(* Logix 5000 project; controller RN21_Architecture 1769-L16ER-BB1B rev 35.11; software revision 35.00; part 3 of 9 *)

ADD_ON_INSTRUCTION AOI_TBC   (* revision 1.0 *)
VAR_INPUT
   FBI_AuditPLC_UID : DINT; {access None, required}
END_VAR
VAR_OUTPUT
   FBO_TBCAuditPLC_UID : DINT; {required}
END_VAR
VAR_INPUT
   FBI_AlarmPLC_UID : DINT; {required}
END_VAR
VAR_OUTPUT
   FBO_TBCAlarmPLC_UID : DINT; {required}
END_VAR
VAR_INPUT
   FBI_RecipePLC_UID : DINT; {required}
END_VAR
VAR_OUTPUT
   FBO_TBCRecipePLC_UID : DINT; {required}
END_VAR
VAR_INPUT
   FBI_UMPLC_UID : DINT; {required}
END_VAR
VAR_OUTPUT
   FBO_TBCUMPLC_UID : DINT; {required}
END_VAR
VAR_INPUT
   FBI_BatchPLC_UID : DINT; {required}
END_VAR
VAR_OUTPUT
   FBO_TBCBatchPLC_UID : DINT; {required}
END_VAR
VAR_INPUT
   FBI_AuditServer_UID : DINT; {required}
END_VAR
VAR_OUTPUT
   FBO_TBCAuditServer_UID : DINT; {required}
END_VAR
VAR_INPUT
   FBI_AlarmServer_UID : DINT; {required}
END_VAR
VAR_OUTPUT
   FBO_TBCAlarmServer_UID : DINT; {required}
END_VAR
VAR_INPUT
   FBI_RecipeServer_UID : DINT; {required}
END_VAR
VAR_OUTPUT
   FBO_TBCRecipeServer_UID : DINT; {required}
END_VAR
VAR_INPUT
   FBI_UMServer_UID : DINT; {required}
END_VAR
VAR_OUTPUT
   FBO_TBCUMServer_UID : DINT; {required}
END_VAR
VAR_INPUT
   FBI_BatchServer_UID : DINT; {required}
END_VAR
VAR_OUTPUT
   FBO_TBCBatchServer_UID : DINT; {required}
   FBO_TBCProcessServer_UID : DINT; {required}
END_VAR
VAR_INPUT
   FBI_ProcessServer_UID : DINT; {required}
   FBI_ProcessPLC_UID : DINT; {required}
END_VAR
VAR_OUTPUT
   FBO_TBCProcessPLC_UID : DINT; {required}
END_VAR
VAR_IN_OUT
   FBIO_Batch_Trigger : BOOL; {required}
   FBIO_UM_Trigger : BOOL; {required}
   FBIO_Process_Trigger : BOOL; {required}
   FBIO_Recipe_Trigger : BOOL; {required}
   FBIO_Audit_Trigger : BOOL; {required}
   FBIO_Alarm_Trigger : BOOL; {required}
END_VAR
VAR_OUTPUT
   FBO_TBCPosition : DINT; {required}
   TBCUID : DINT; {required}
END_VAR
VAR_IN_OUT
   FBI_TBCServerAlarm_Trig : BOOL; {required}
   FBI_TBCServerProces_Trig : BOOL; {required}
   FBI_TBCServerAudit_Trig : BOOL; {required}
   FBI_TBCServerBatch_Trig : BOOL; {required}
   FBI_TBCServerRecipe_Trig : BOOL; {required}
   FBI_TBCServerUM_Trig : BOOL; {required}
END_VAR
VAR
   TMR_TBCTrigger : TIMER := (PRE := 60000); {access None}
   CTU_TBCUID : COUNTER := (PRE := 32767); {access None}
   FBL_TBCPosition : DINT; {access None}
   TMRTBC_AlmTrigRst : TIMER := (PRE := 10000); {access None}
   TMRTBC_UMTrigRst : TIMER := (PRE := 10000); {access None}
   TMRTBC_ProcessTrigRst : TIMER := (PRE := 10000); {access None}
   TMRTBC_AuditTrigRst : TIMER := (PRE := 10000); {access None}
   TMRTBC_BatchTrigRst : TIMER := (PRE := 10000); {access None}
   TMRTBC_RecipeTrigRst : TIMER := (PRE := 10000); {access None}
END_VAR

ROUTINE Logic   (* ladder *)
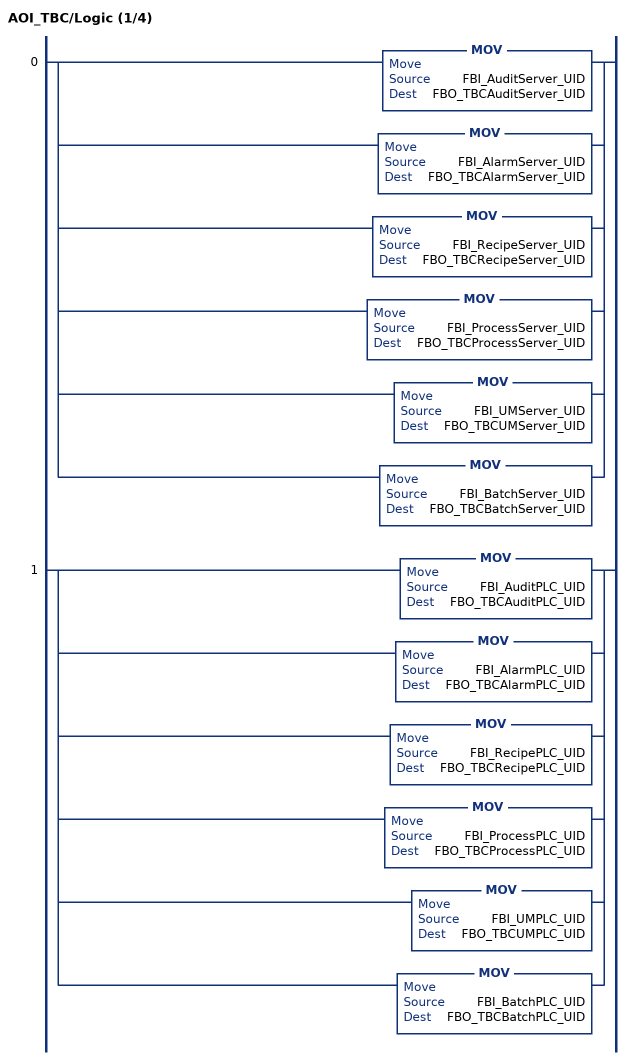
   0: [MOV(FBI_AuditServer_UID,FBO_TBCAuditServer_UID) ,MOV(FBI_AlarmServer_UID,FBO_TBCAlarmServer_UID) ,MOV(FBI_RecipeServer_UID,FBO_TBCRecipeServer_UID) ,MOV(FBI_ProcessServer_UID,FBO_TBCProcessServer_UID) ,MOV(FBI_UMServer_UID,FBO_TBCUMServer_UID) ,MOV(FBI_BatchServer_UID,FBO_TBCBatchServer_UID) ];
   1: [MOV(FBI_AuditPLC_UID,FBO_TBCAuditPLC_UID) ,MOV(FBI_AlarmPLC_UID,FBO_TBCAlarmPLC_UID) ,MOV(FBI_RecipePLC_UID,FBO_TBCRecipePLC_UID) ,MOV(FBI_ProcessPLC_UID,FBO_TBCProcessPLC_UID) ,MOV(FBI_UMPLC_UID,FBO_TBCUMPLC_UID) ,MOV(FBI_BatchPLC_UID,FBO_TBCBatchPLC_UID) ];
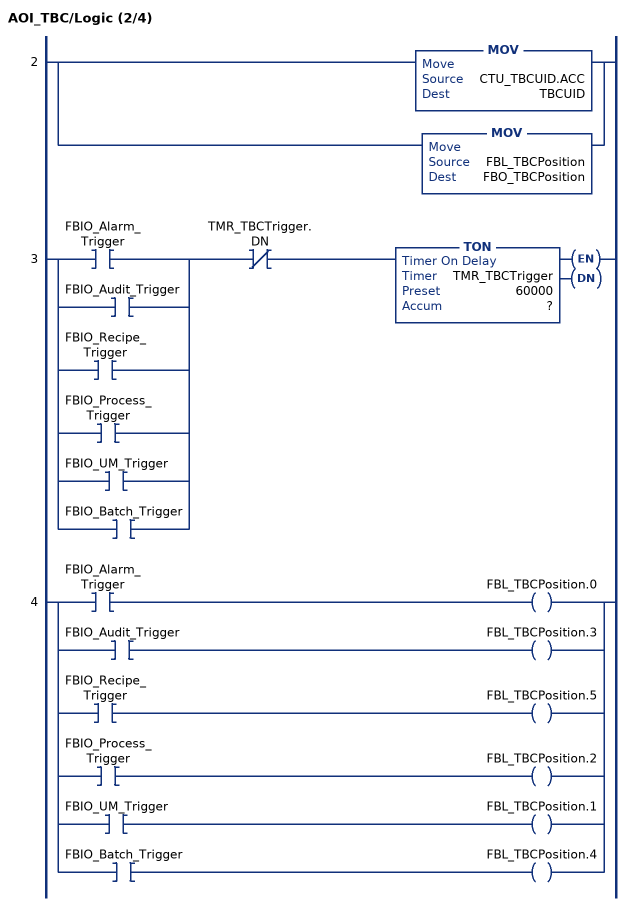
   2: [MOV(CTU_TBCUID.ACC,TBCUID) ,MOV(FBL_TBCPosition,FBO_TBCPosition) ];
   3: [XIC(FBIO_Alarm_Trigger) ,XIC(FBIO_Audit_Trigger) ,XIC(FBIO_Recipe_Trigger) ,XIC(FBIO_Process_Trigger) ,XIC(FBIO_UM_Trigger) ,XIC(FBIO_Batch_Trigger) ]XIO(TMR_TBCTrigger.DN)TON(TMR_TBCTrigger,?,?);
   4: [XIC(FBIO_Alarm_Trigger) OTE(FBL_TBCPosition.0) ,XIC(FBIO_Audit_Trigger) OTE(FBL_TBCPosition.3) ,XIC(FBIO_Recipe_Trigger) OTE(FBL_TBCPosition.5) ,XIC(FBIO_Process_Trigger) OTE(FBL_TBCPosition.2) ,XIC(FBIO_UM_Trigger) OTE(FBL_TBCPosition.1) ,XIC(FBIO_Batch_Trigger) OTE(FBL_TBCPosition.4) ];
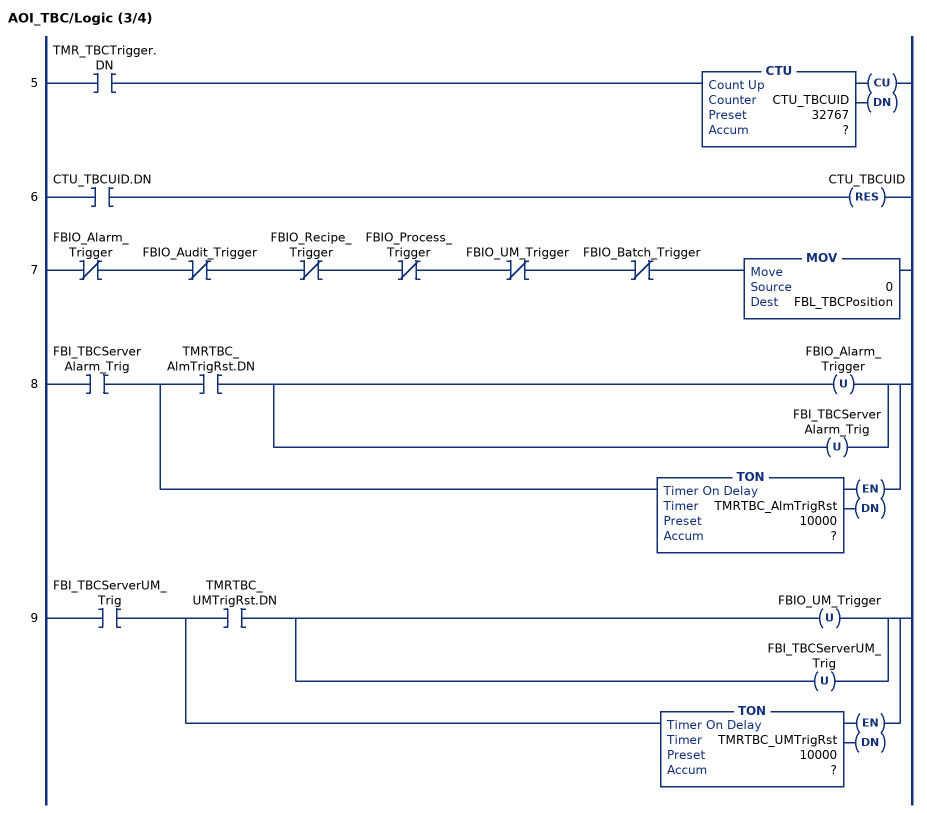
   5: XIC(TMR_TBCTrigger.DN)CTU(CTU_TBCUID,?,?);
   6: XIC(CTU_TBCUID.DN)RES(CTU_TBCUID);
   7: XIO(FBIO_Alarm_Trigger)XIO(FBIO_Audit_Trigger)XIO(FBIO_Recipe_Trigger)XIO(FBIO_Process_Trigger)XIO(FBIO_UM_Trigger)XIO(FBIO_Batch_Trigger)MOV(0,FBL_TBCPosition);
   8: XIC(FBI_TBCServerAlarm_Trig)[XIC(TMRTBC_AlmTrigRst.DN) [OTU(FBIO_Alarm_Trigger) ,OTU(FBI_TBCServerAlarm_Trig) ] ,TON(TMRTBC_AlmTrigRst,?,?) ];
   9: XIC(FBI_TBCServerUM_Trig)[XIC(TMRTBC_UMTrigRst.DN) [OTU(FBIO_UM_Trigger) ,OTU(FBI_TBCServerUM_Trig) ] ,TON(TMRTBC_UMTrigRst,?,?) ];
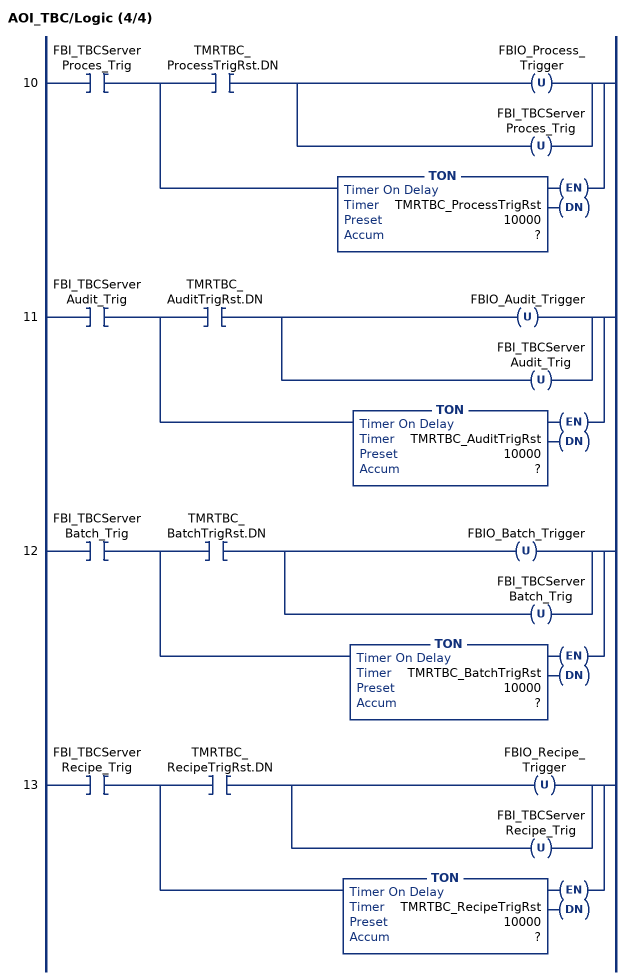
   10: XIC(FBI_TBCServerProces_Trig)[XIC(TMRTBC_ProcessTrigRst.DN) [OTU(FBIO_Process_Trigger) ,OTU(FBI_TBCServerProces_Trig) ] ,TON(TMRTBC_ProcessTrigRst,?,?) ];
   11: XIC(FBI_TBCServerAudit_Trig)[XIC(TMRTBC_AuditTrigRst.DN) [OTU(FBIO_Audit_Trigger) ,OTU(FBI_TBCServerAudit_Trig) ] ,TON(TMRTBC_AuditTrigRst,?,?) ];
   12: XIC(FBI_TBCServerBatch_Trig)[XIC(TMRTBC_BatchTrigRst.DN) [OTU(FBIO_Batch_Trigger) ,OTU(FBI_TBCServerBatch_Trig) ] ,TON(TMRTBC_BatchTrigRst,?,?) ];
   13: XIC(FBI_TBCServerRecipe_Trig)[XIC(TMRTBC_RecipeTrigRst.DN) [OTU(FBIO_Recipe_Trigger) ,OTU(FBI_TBCServerRecipe_Trig) ] ,TON(TMRTBC_RecipeTrigRst,?,?) ];
END_ROUTINE
END_ADD_ON_INSTRUCTION

VAR_GLOBAL   (* controller tags *)
   ALM_TriggerId : BOOL := 1;
   ALM_UniqueNum : DINT := 300;
   ALMSer : UDT_Alarm := (ALM_YearValue := 2026, ALM_MonthValue := 3, ALM_DayValue := 3, ALM_HourValue := 18, ALM_MinuteValue := 48, ALM_SecondValue := 11, ALM_AlarmId1 := 3);
   AUD_TriggerId : BOOL;
   AUD_UniqueNum : DINT := 911;
   AUDSer : UDT_Audit := (AUD_YearValue := 2026, AUD_MonthValue := 3, AUD_DayValue := 3, AUD_HourValue := 12, AUD_SecondValue := 30, AUD_ActionId := 6009, AUD_NewValue := 389.0, AUD_AppUserId := 'EMGUSER');
   BACK_BATCH_NO : STRING := 'ee3';
   BACK_BatchStartACK : DINT;
   BACK_LOT_NO : STRING := 'uuuu';
   BMAN_BatchUniqueId : DINT := 63;
   BMAN_TriggerBit : BOOL;
   BMANSer : UDT_Batch := (BMAN_YearValue := 2026, BMAN_MonthValue := 3, BMAN_DayValue := 2, BMAN_HourValue := 17, BMAN_MinuteValue := 33, BMAN_SecondValue := 37, BMAN_BatchStatus := 2, BMAN_BATCH_RECIPENAME := 'CLST5000', BMAN_LOT_NO := 'lot1', BMAN_PRODUCT_CODE := 'Compa', BMAN_PRODUCT_NAME := 'Compa', BMAN_BATCH_NO := 'Tes');
   Controller_FirstScan : BOOL;
   DummyBit : BOOL;
   EmergencyLoginActivated_Bit : BOOL := 1;
   EmergencyUserIDEqual : BOOL;
   EmergencyUserPaswdEqual : BOOL;
   FCI_C1PAUSE_RELEASE : BOOL;
   FCI_C1START : BOOL;
   FCI_C1STOP : BOOL;
   FCO_C1STARTED : BOOL;
   HB_HEART_BEAT : BOOL := 1;
   LBSer : UDT_Login := (LOGIN_YearValue := 2026, LOGIN_MonthValue := 3, LOGIN_DayValue := 4, LOGIN_HourValue := 10, LOGIN_MinuteValue := 9, LOGIN_SecondValue := 53, LOGIN_Reason := 28, LOGIN_LoginReason := -1, LOGIN_AppUserId := 'Navin$00$00');
   LOGIN_TriggerId : BOOL := 1;
   LOGIN_UniqueNum : DINT := 570;
   PDL_Trigger : BOOL;
   PDL_UID : DINT := 701;
   PDLSer : UDT_Process := (PDL_Year := 2026, PDL_Month := 1, PDL_Date := 13, PDL_Hour := 17, PDL_Minute := 22, PDL_Second := 27, PDL_CYCLEID := 2, PDL_ProcessData[0] := 3.0, PDL_ProcessData[1] := 5.0, PDL_ProcessData[2] := 5.0, PDL_ProcessData[3] := 6.0, PDL_ProcessData[4] := 2.2, PDL_ProcessData[5] := 11.2, PDL_ProcessData[6] := 11.9, PDL_ProcessData[7] := 41.5);
   RM_RecipeAck : DINT := 2;
   RM_RecipeCode : STRING := 'CLST5000';
   RN21_BACK_BatchSize : REAL := 51.02;
   RN21_BACK_ProductCode : STRING := 'AKHBJ';
   RN21_BACK_ProductName : STRING := 'AEBJH';
   RN21_EmgUserID : STRING := 'EMGUSER';
   RN21_FirstScan : BOOL;
   RN21_HMIScrennControl : DINT;
   RN21_PDLMainONS : BOOL;
   RN21_UM_EmgPSWD : STRING := 'EMG1234';
   RP_Trigger : BOOL;
   RP_UID : DINT := 31;
   RPSer : UDT_Recipe := (RP_Year := 2026, RP_Month := 1, RP_Date := 12, RP_Hour := 10, RP_Minute := 57, RP_Second := 54, RP_RecipeData1[0] := 10.0, RP_RecipeData1[1] := 11.1, RP_RecipeData1[2] := 22.2, RP_RecipeData1[3] := 33.3, RP_RecipeData1[4] := 44.4, RP_RecipeData1[5] := 55.5, RP_RecipeData1[6] := 66.6, RP_RecipeData1[7] := 77.7, RP_RecipeData1[8] := 88.8, RP_RecipeData1[9] := 99.9, RP_RecipeData2[0] := 10, RP_RecipeData2[1] := 20, RP_RecipeData2[2] := 30, RP_RecipeData2[3] := 40, RP_RecipeData2[4] := 50, RP_RecipeData2[5] := 60, RP_RecipeData2[6] := 70, RP_RecipeData2[7] := 80, RP_RecipeData2[8] := 90, RP_RecipeData2[9] := 100);
   RTC_DATE_AND_TIME_UNLATCH_DELAY : COUNTER := (PRE := 2);
   RTC_DAY : DINT := 3;
   RTC_HOUR : DINT := 12;
   RTC_MINUTE : DINT := 23;
   RTC_MONTH : DINT := 3;
   RTC_SAVE_DATE_AND_TIME : BOOL;
   RTC_SECONDS : DINT := 14;
   RTC_UniqueId : DINT := 97;
   RTC_YEAR : DINT := 2026;
   ServerRTC : DINT[8] := ([0] := 2026, [1] := 3, [2] := 25, [3] := 5, [4] := 43, [5] := 2);
   TBC_ALARMBLOCK_PLCUID : DINT := 304;
   TBC_ALARMBLOCK_SERVERUID : DINT := 300;
   TBC_ALARMBLOCK_TRIGGER : BOOL;
   TBC_AUDITBLOCK_PLCUID : DINT := 911;
   TBC_AUDITBLOCK_SERVERUID : DINT := 911;
   TBC_AUDITBLOCK_TRIGGER : BOOL;
   TBC_BATCHMGMTBLOCK_PLCUID : DINT;
   TBC_BATCHMGMTBLOCK_SERVERUID : DINT := 63;
   TBC_BATCHMGMTBLOCK_TRIGGER : BOOL;
   TBC_POSITION : DINT := 3;
   TBC_PROCESSBLOCK_PLCUID : DINT := 701;
   TBC_PROCESSBLOCK_SERVERUID : DINT := 701;
   TBC_PROCESSBLOCK_TRIGGER : BOOL;
   TBC_RECIPEBLOCK_PLCUID : DINT := 31;
   TBC_RECIPEBLOCK_SERVERUID : DINT := 31;
   TBC_RECIPEBLOCK_TRIGGER : BOOL;
   TBC_UID : DINT;
   TBC_UMBLOCK_PLCUID : DINT := 581;
   TBC_UMBLOCK_SERVERUID : DINT := 570;
   TBC_UMBLOCK_TRIGGER : BOOL;
   UM_ACT : DINT;
   UM_Confirmation_Bit : BOOL;
   UM_EXPIRY : DINT;
   UM_EXPIRY_DAYS : DINT := 78;
   UM_lockoutDurationLeft : DINT;
   UM_LVL : DINT;
   UM_NoOfAttempts : DINT := 5;
   UM_PWD : STRING := '0';
   UM_Status : DINT;
   UM_UID : STRING := '0';
   UM_UID_OUT : STRING := 'Navin';
   UM_UniqueID : DINT := 520;
END_VAR

PROGRAM MainProgram   (* main routine MainRoutine *)
VAR
   ALMSrc : UDT_Alarm := (ALM_YearValue := 2026, ALM_MonthValue := 3, ALM_DayValue := 4, ALM_HourValue := 14, ALM_MinuteValue := 57, ALM_SecondValue := 10, ALM_AlarmId1 := 1);
   ALMSrc_UniqueNum : DINT := 304;
   ANM_C1Pause_Release : BOOL;
   ANM_C1StartReq : BOOL;
   ANM_C1StopReq_Auto : BOOL;
   ANM_C1StopReq_HMI : BOOL;
   ANM_C2Pause_Release : BOOL;
   ANM_C2StartReq : BOOL;
   ANM_C2StopReq_Auto : BOOL;
   ANM_C2StopReq_HMI : BOOL;
   ANM_C3Pause_Release : BOOL;
   ANM_C3StartReq : BOOL;
   ANM_C3StopReq_Auto : BOOL;
   ANM_C3StopReq_HMI : BOOL;
   ANM_C4Pause_Release : BOOL;
   ANM_C4StartReq : BOOL;
   ANM_C4StopReq_Auto : BOOL;
   ANM_C4StopReq_HMI : BOOL;
   ANM_C5Pause_Release : BOOL;
   ANM_C5StartReq : BOOL;
   ANM_C5StopReq_Auto : BOOL;
   ANM_C5StopReq_HMI : BOOL;
   ANM_CStopReq_Alarm : BOOL;
   ANM_CycleReset : BOOL;
   AUDSrc : UDT_Audit := (AUD_YearValue := 2026, AUD_MonthValue := 3, AUD_DayValue := 4, AUD_HourValue := 14, AUD_MinuteValue := 57, AUD_SecondValue := 10, AUD_ActionId := 6009, AUD_NewValue := 389.0, AUD_AppUserId := 'EMGUSER');
   AUDSrc_UniqueNum : DINT := 911;
   BIT_RESET_TMR : TIMER := (PRE := 5000);
   BMANSrc : UDT_Batch := (BMAN_YearValue := 2026, BMAN_MonthValue := 3, BMAN_DayValue := 4, BMAN_HourValue := 14, BMAN_MinuteValue := 57, BMAN_SecondValue := 10, BMAN_BatchStatus := 2, BMAN_BATCH_RECIPENAME := 'CLS');
   BMANSrc_UniqueNum : DINT := 63;
   Delformovingupdatedtimertonewpswd : TIMER := (PRE := 2000);
   EmgLoginDn : BOOL;
   EnableInactivity : DINT;
   ExpDays_NoofattemptsLeft_visb : BOOL;
   ExpDays_NoofattemptsLeft_visbility : BOOL := 1;
   ExpiryDays_MovFrmSrv : DINT := 78;
   FC_ALM_Arch : AOI_ALM_Arch := (FBI_PLCServerCommFailed := 1);
   FC_ALM_DC : AOI_ALM_DataCapture[160] := ([0].FBI_AlarmTag := 1, [0].FBO_AlarmPosID := 1);
   FC_AUD_Arch : AOI_AUD_Arch := (FBI_PLCServerCommFailed := 1);
   FC_BMAN_Arch : AOI_BMAN_Arch := (FBI_PLCServerCommFailed := 1);
   FC_LB_Arch : AOI_LOGIN_Arch := (FBI_PLCServerCommFailed := 1);
   FC_PDL_Arch : AOI_PDL_Arch := (FBI_PLCServerCommFailed := 1);
   FC_PDL_DC : AOI_PDL_DataCapture[10] := ([0].FBI_IsPrintIntervalReq := 1, [0].FBI_PrintInterval := 60, [0].FBI_OneSecTrig := 1, [0].FBI_Enable := 1, [0].FBO_Active := 1, [1].FBI_IsPrintIntervalReq := 1, [1].FBI_PrintInterval := 60, [1].FBI_OneSecTrig := 1, [1].FBI_Enable := 1, [1].FBO_Active := 1, [2].FBI_IsPrintIntervalReq := 1, [2].FBI_PrintInterval := 60, [2].FBI_OneSecTrig := 1, [2].FBI_Enable := 1, [2].FBO_Active := 1, [3].FBI_IsPrintIntervalReq := 1, [3].FBI_PrintInterval := 60, [3].FBI_OneSecTrig := 1, [3].FBI_Enable := 1, [3].FBO_Active := 1, [4].FBI_IsPrintIntervalReq := 1, [4].FBI_PrintInterval := 60, [4].FBI_OneSecTrig := 1, [4].FBI_Enable := 1, [4].FBO_Active := 1);
   FC_RP_Arch : AOI_RP_Arch := (FBI_PLCServerCommFailed := 1);
   FC_TBC : AOI_TBC := (FBI_AuditPLC_UID := 911, FBO_TBCAuditPLC_UID := 911, FBI_AlarmPLC_UID := 304, FBO_TBCAlarmPLC_UID := 304, FBI_RecipePLC_UID := 31, FBO_TBCRecipePLC_UID := 31, FBI_UMPLC_UID := 581, FBO_TBCUMPLC_UID := 581, FBI_BatchPLC_UID := 63, FBO_TBCBatchPLC_UID := 63, FBI_AuditServer_UID := 911, FBO_TBCAuditServer_UID := 911, FBI_AlarmServer_UID := 300, FBO_TBCAlarmServer_UID := 300, FBI_RecipeServer_UID := 31, FBO_TBCRecipeServer_UID := 31, FBI_UMServer_UID := 570, FBO_TBCUMServer_UID := 570, FBI_BatchServer_UID := 63, FBO_TBCBatchServer_UID := 63, FBO_TBCProcessServer_UID := 701, FBI_ProcessServer_UID := 701, FBI_ProcessPLC_UID := 701, FBO_TBCProcessPLC_UID := 701, FBO_TBCPosition := 3, TBCUID := 2932);
   FCI_ALARM : BOOL;
   FCI_AlarmReset : BOOL;
   FCI_ALMDataLogTrig : BOOL;
   FCI_AUDDataLogTrig : BOOL;
   FCI_BMANDataLogTrig : BOOL;
   FCI_C1COMPLETED : BOOL;
   FCI_C2COMPLETED : BOOL;
   FCI_C2PAUSE_RELEASE : BOOL;
   FCI_C2START : BOOL;
   FCI_C2STOP : BOOL;
   FCI_C3COMPLETED : BOOL;
   FCI_C3PAUSE_RELEASE : BOOL;
   FCI_C3START : BOOL;
   FCI_C3STOP : BOOL;
   FCI_C4COMPLETED : BOOL;
   FCI_C4PAUSE_RELEASE : BOOL;
   FCI_C4START : BOOL;
   FCI_C4STOP : BOOL;
   FCI_C5COMPLETED : BOOL;
   FCI_C5PAUSE_RELEASE : BOOL;
   FCI_C5STARTED : BOOL;
   FCI_C5STOP : BOOL;
   FCI_LBDataLogTrig : BOOL;
   FCI_PDLDataLogTrig : BOOL;
   FCI_PrintInterval : INT := 60;
   FCI_PROCESSRESET : BOOL;
   FCI_RPDataLogTrig : BOOL;
   FCO_ALMTrig : DINT[5];
   FCO_C1CMPLTSTSMOVTRIG : BOOL;
   FCO_C1PAUSED : BOOL;
   FCO_C1PAUSEDSTSMOVTRIG : BOOL;
   FCO_C1RELEASEDSTSMOVTRIG : BOOL;
   FCO_C1RUNNINGSTSMOVTRIG : BOOL;
   FCO_C1STOPEDALMSTSMOVTRIG : BOOL;
   FCO_C1STOPEDSTSMOVTRIG : BOOL;
   FCO_C2CMPLTSTSMOVTRIG : BOOL;
   FCO_C2PAUSED : BOOL;
   FCO_C2PAUSEDSTSMOVTRIG : BOOL;
   FCO_C2RELEASEDSTSMOVTRIG : BOOL;
   FCO_C2RUNNINGSTSMOVTRIG : BOOL;
   FCO_C2STARTED : BOOL;
   FCO_C2STOPEDALMSTSMOVTRIG : BOOL;
   FCO_C2STOPEDSTSMOVTRIG : BOOL;
   FCO_C3CMPLTSTSMOVTRIG : BOOL;
   FCO_C3PAUSED : BOOL;
   FCO_C3PAUSEDSTSMOVTRIG : BOOL;
   FCO_C3RELEASEDSTSMOVTRIG : BOOL;
   FCO_C3RUNNINGSTSMOVTRIG : BOOL;
   FCO_C3STARTED : BOOL;
   FCO_C3STOPEDALMSTSMOVTRIG : BOOL;
   FCO_C3STOPEDSTSMOVTRIG : BOOL;
   FCO_C4CMPLTSTSMOVTRIG : BOOL;
   FCO_C4PAUSED : BOOL;
   FCO_C4PAUSEDSTSMOVTRIG : BOOL;
   FCO_C4RELEASEDSTSMOVTRIG : BOOL;
   FCO_C4RUNNINGSTSMOVTRIG : BOOL;
   FCO_C4STARTED : BOOL;
   FCO_C4STOPEDALMSTSMOVTRIG : BOOL;
   FCO_C4STOPEDSTSMOVTRIG : BOOL;
   FCO_C5CMPLTSTSMOVTRIG : BOOL;
   FCO_C5PAUSED : BOOL;
   FCO_C5PAUSEDSTSMOVTRIG : BOOL;
   FCO_C5RELEASEDSTSMOVTRIG : BOOL;
   FCO_C5RUNNINGSTSMOVTRIG : BOOL;
   FCO_C5STARTED : BOOL;
   FCO_C5STOPEDALARMSTSMOVTRIG : BOOL;
   FCO_C5STOPEDSTSMOVTRIG : BOOL;
   HMI_ChangePswd : BOOL;
   HMI_CONTROL_SCREEN : DINT;
   HmiCurrentScreen : DINT;
   HMIOLDSCREENVALUE : DINT;
   HMISCREEN : BOOL;
   HMISCREENCHANGED : BOOL;
   inactivity_in_minutes : DINT;
   inactivity_time : DINT := 5;
   INTERNAL_RN21_HB_PLC2ServerCommFailed : BOOL;
   INTERNAL_RN21_PLC2HMICommFailed : BOOL;
   InvalidBit : BOOL;
   LBSrc : UDT_Login := (LOGIN_YearValue := 2026, LOGIN_MonthValue := 3, LOGIN_DayValue := 4, LOGIN_HourValue := 14, LOGIN_MinuteValue := 57, LOGIN_SecondValue := 10, LOGIN_Reason := -1, LOGIN_LoginReason := -32768, LOGIN_AppUserId := 'EMGUSER');
   LBSrc_UniqueNum : DINT := 581;
   Lockout_Visb : BOOL;
   Logged_User : STRING := '0';
   LoginDNDel : TIMER := (PRE := 5000);
   MaskTag : STRING := '************';
   MaskTag1 : STRING := '0';
   New_Pswd : STRING := '0';
   New_Pswd_mask : STRING := '************';
   New_Pswd_mask1 : STRING := '0';
   Password_Change_Yes_Button_In_HMI : BOOL;
   PDLSrc : UDT_Process := (PDL_Year := 2026, PDL_Month := 3, PDL_Date := 4, PDL_Hour := 14, PDL_Minute := 57, PDL_Second := 10, PDL_CYCLEID := 2, PDL_ProcessData[0] := 3.0, PDL_ProcessData[1] := 5.0, PDL_ProcessData[2] := 5.0, PDL_ProcessData[3] := 6.0, PDL_ProcessData[4] := 2.2, PDL_ProcessData[5] := 11.2, PDL_ProcessData[6] := 11.9, PDL_ProcessData[7] := 41.5);
   PDLSrc_PDL_UID : DINT := 701;
   PLC_HMI_CommTag : BOOL;
   PLC_RTC : DINT[7] := ([0] := 2026, [1] := 3, [2] := 4, [3] := 14, [4] := 57, [5] := 10, [6] := 68182);
   PrintIntervalReq : BOOL := 1;
   Pswd_UpadatedSuccessfully : BOOL;
   pwdons : BOOL;
   RecipeEntryFloat : REAL[20] := ([0] := 10.0, [1] := 11.1, [2] := 22.2, [3] := 33.3, [4] := 44.4, [5] := 55.5, [6] := 66.6, [7] := 77.7, [8] := 88.8, [9] := 99.9, [10] := 100.0, [11] := 111.1, [12] := 222.2, [13] := 333.3, [14] := 444.4, [15] := 555.5, [16] := 666.6, [17] := 777.7, [18] := 888.8, [19] := 12.2);
   RecipeEntryInt : INT[11] := ([0] := 10, [1] := 20, [2] := 30, [3] := 40, [4] := 50, [5] := 60, [6] := 70, [7] := 80, [8] := 90, [9] := 100, [10] := 110);
   Remaining_time : DINT;
   remaining_time_compareTag : DINT;
   RN21_AUD_BAMTrig : DINT[5];
   RN21_AUD_BAT_NTrig : DINT[4];
   RN21_AUD_BAT_PTrig : DINT[4];
   RN21_AUD_CompVal : REAL[305] := ([0] := 350.0, [1] := 700.0, [2] := 360.0, [3] := 61.0, [4] := 893.0, [5] := 183.0, [6] := 947.0, [7] := 317.0, [8] := 412.0, [9] := 389.0);
   RN21_AUD_HoldVal : REAL[305] := ([0] := 300.0, [1] := 600.0);
   RN21_AUD_NE_ONS : BOOL[320];
   RN21_AUD_NEG_ONS : BOOL[128];
   RN21_AUD_NETrig : DINT[11];
   RN21_AUD_POS_ONS : BOOL[128];
   RN21_AUDBAM_ONS : BOOL[128];
   RN21_AutoLogedOut : BOOL;
   RN21_BACK_BatchDataStatus : BOOL;   // BATCH START ACKNOWLEDGEMENT STATUS FROM SERVER
   RN21_BACK_BatchStartHMI : BOOL;   // HMI BATCH START IN BATCH DETAILS
   RN21_BACKONS : DINT[1];
   RN21_BMAN_BatchStarted : BOOL;   // BATCH STARTED IN BATCH MANAGEMENT
   RN21_BMAN_BatchStopped : BOOL;   // BATCH STOPPED IN BATCH MANAGEMENT
   RN21_BMAN_HMIBatchStart : BOOL;   // BATCH START
   RN21_BMAN_HMIBatchStop : BOOL;
   RN21_BMANBASTPNEG : BOOL;
   RN21_BMANBASTPPOS : BOOL;
   RN21_BMANBASTRTNEG : BOOL;
   RN21_BMANBASTRTPOS : BOOL;
   RN21_DC_Active : BOOL := 1;
   RN21_DC_Enable : BOOL := 1;
   RN21_HB_PLC2ServerCommFailed : BOOL := 1;
   RN21_LBONS : DINT[2];
   RN21_LBStatus : INT := -1;   // Login Block Status
   RN21_LBStatus1 : DINT;
   RN21_Map_BAM : BOOL[128];
   RN21_Map_BAT : BOOL[32];
   RN21_Map_NE : REAL[350] := ([0] := 350.0, [1] := 700.0, [2] := 360.0, [3] := 61.0, [4] := 893.0, [5] := 183.0, [6] := 947.0, [7] := 317.0, [8] := 412.0, [9] := 389.0);
   RN21_MapBAT_OB : BOOL[128];
   RN21_MapBAT_SB : BOOL[128];
   RN21_PDL_OSTBit : BOOL;
   RN21_PDL_OSTTempInt : DINT := 9;   // One Second Trig
   RN21_PDLMAPONS : DINT;
   RN21_PDLParam : REAL[20] := ([0] := 3.0, [1] := 5.0, [2] := 5.0, [3] := 6.0, [4] := 2.2, [5] := 11.2, [6] := 11.9, [7] := 41.5);
   RN21_PDLStatus : DINT := 2;
   RN21_PDLTrig : DINT;
   RN21_PLC2HMICommFailed : BOOL;
   RN21_PrintInterval : DINT := 60;
   RN21_RM_BITRESET : BOOL;
   RN21_RM_HMICheck : BOOL;
   RN21_RM_HMICODE : STRING := 'CLST5000';
   RN21_RM_HMILoad : BOOL;
   RN21_RM_LOADBIT : BOOL;
   RN21_RM_LOADBTNVISB : BOOL := 1;
   RN21_RM_LOADDLY_TMRBIT : BOOL;
   RN21_RM_LOADDLYBIT : BOOL;
   RN21_RM_LOADSTATUS : DINT := 1;
   RN21_RM_LOADVISB : BOOL;
   RN21_RM_ONS : BOOL[64];
   RN21_RM_STATUS_VISB : BOOL := 1;
   RN21_Test_BAM : BOOL[128];
   RN21_Test_BAT : BOOL[128];
   RN21_TEST_NE : DINT[350];
   RN21_UM_ActiveUserMovFrmSrv : DINT := 1;
   RN21_UM_Empty : STRING := '0';   // Whenever Logout Will happen moving the Empty
   RN21_UM_ExpiryBitMovFrmSrv : DINT;
   RN21_UM_HMIPSWD_Visb : BOOL;
   RN21_UM_HMIPSWDAPPLY : BOOL;
   RN21_UM_HMIUserIDApply : BOOL;
   RN21_UM_HMIUSERPSWD : STRING := '0';
   RN21_UM_INVALIDUserLatch : BOOL;
   RN21_UM_MaintBit : BOOL;
   RN21_UM_OperBit : BOOL;
   RN21_UM_Status_Visb : BOOL := 1;
   RN21_UM_SupBit : BOOL;
   RN21_UM_USERIDEquLatch : BOOL;
   RN21_UM_USERIDMovFrmSrv : STRING := 'saira';
   RN21_UM_USERIDNotEqual : BOOL;
   RN21_UM_UserLogout : BOOL;
   RN21_UM_UserLvlMovFrmSrv : DINT;
   RN21_UMAdmBit : BOOL;
   RN21_UMLogoutTag : INT;
   RN21_UMONS : DINT := 16;
   RN21_UserLoginDN : BOOL;
   RP_Param2 : DINT := 10;
   RPSrc : UDT_Recipe := (RP_Year := 2026, RP_Month := 3, RP_Date := 4, RP_Hour := 14, RP_Minute := 57, RP_Second := 10, RP_RecipeData1[5] := 55.5, RP_RecipeData1[6] := 66.6, RP_RecipeData1[7] := 77.7, RP_RecipeData1[8] := 88.8, RP_RecipeData1[9] := 99.9, RP_RecipeData2[5] := 60, RP_RecipeData2[6] := 70, RP_RecipeData2[7] := 80, RP_RecipeData2[8] := 90, RP_RecipeData2[9] := 100);
   RPSrc_RP_UID : DINT := 31;
   RTC_DATE_AND_TIME_UNLATCH_DELAY1 : TIMER := (PRE := 2000);
   Temp_int : DINT := 7;
   teset : BOOL;
   TestAlarmTag : BOOL[160];
   TestProcessTag : REAL[8] := ([0] := 3.0, [1] := 5.0, [2] := 5.0, [3] := 6.0, [4] := 2.2, [5] := 11.2, [6] := 11.9, [7] := 41.5);
   TMR_AutoLogout : TIMER := (PRE := 300000);
   TMR_AutoLogoutRstDly : TIMER := (PRE := 6000);
   TMR_BatchStartAckDlyRst : TIMER := (PRE := 2000);
   TMR_BatchStrtdDlyStsMov : TIMER := (PRE := 2000);
   TMR_HBSetDelay : TIMER := (PRE := 2000);
   TMR_LOAD_DLY : TIMER := (PRE := 30000);
   TMR_LOGOUT : TIMER := (PRE := 50);
   TMR_LogoutTagRst : TIMER := (PRE := 5000);
   TMR_ONE_SECBIT_RST : TIMER := (PRE := 500);
   TMR_PHSetDelay : TIMER := (PRE := 500, ACC := 500, EN := 1, DN := 1);
   TMR_PLCtoHMICommCheck : TIMER := (PRE := 30000);
   TMR_PLCToSrvComCheck : TIMER := (PRE := 120000, ACC := 120002, EN := 1, DN := 1);
   TMR_SvrConfrm_BIT : TIMER := (PRE := 2000);
   TMR_UMLogoutTag : TIMER := (PRE := 180000);
   TMR_UserIDRstDly : TIMER := (PRE := 1000);
   TMRHMIPSWDVisb_Dly : TIMER;
   True : BOOL := 1;
   UM_LogGenDelay : TIMER := (PRE := 500);
   UM_Status1 : DINT;
END_VAR
VAR {public}
   PDL_Para1 : REAL := 3.0;
   PDL_Para2 : REAL := 5.0;
   PDL_Para3 : REAL := 5.0;
   PDL_Para4 : REAL := 6.0;
   RM_Param1 : DINT;
   RM_Param10 : REAL;
   RM_Param2 : DINT;
   RM_Param3 : DINT;
   RM_Param4 : DINT;
   RM_Param5 : DINT;
   RM_Param6 : REAL;
   RM_Param7 : REAL;
   RM_Param8 : REAL;
   RM_Param9 : REAL;
   RP_Param1 : DINT := 10;
   RP_Param10 : REAL := 44.4;
   RP_Param3 : DINT := 10;
   RP_Param4 : DINT := 10;
   RP_Param5 : DINT := 10;
   RP_Param6 : REAL := 10.0;
   RP_Param7 : REAL := 11.1;
   RP_Param8 : REAL := 22.2;
   RP_Param9 : REAL := 33.3;
END_VAR

ROUTINE MainRoutine   (* ladder *)
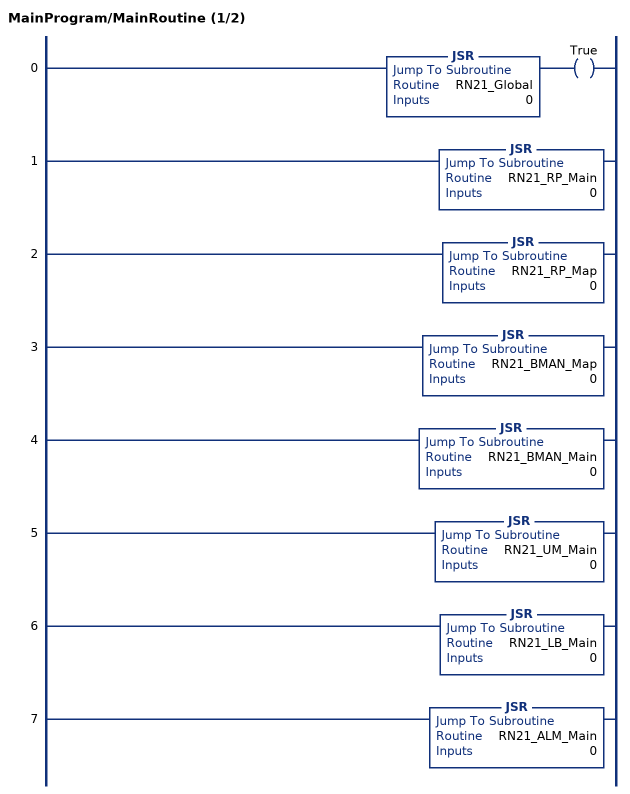
   0: JSR(RN21_Global,0)OTE(True);
   1: JSR(RN21_RP_Main,0);
   2: JSR(RN21_RP_Map,0);
   3: JSR(RN21_BMAN_Map,0);
   4: JSR(RN21_BMAN_Main,0);
   5: JSR(RN21_UM_Main,0);
   6: JSR(RN21_LB_Main,0);
   7: JSR(RN21_ALM_Main,0);
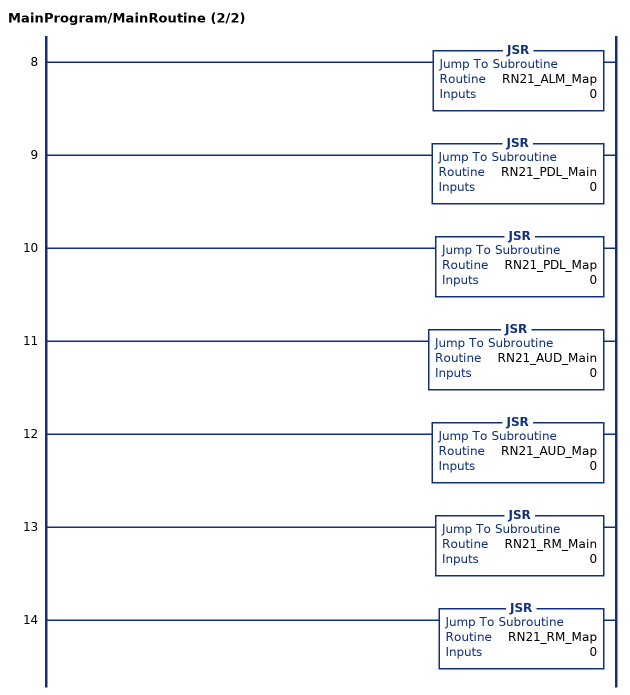
   8: JSR(RN21_ALM_Map,0);
   9: JSR(RN21_PDL_Main,0);
   10: JSR(RN21_PDL_Map,0);
   11: JSR(RN21_AUD_Main,0);
   12: JSR(RN21_AUD_Map,0);
   13: JSR(RN21_RM_Main,0);
   14: JSR(RN21_RM_Map,0);
END_ROUTINE

ROUTINE RN21_ALM_Main   (* ladder *)
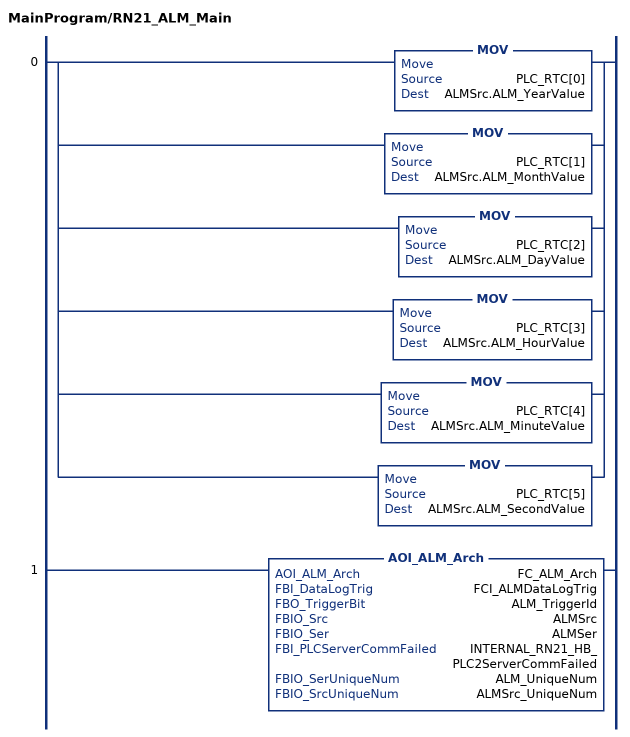
   0: [MOV(PLC_RTC[0],ALMSrc.ALM_YearValue) ,MOV(PLC_RTC[1],ALMSrc.ALM_MonthValue) ,MOV(PLC_RTC[2],ALMSrc.ALM_DayValue) ,MOV(PLC_RTC[3],ALMSrc.ALM_HourValue) ,MOV(PLC_RTC[4],ALMSrc.ALM_MinuteValue) ,MOV(PLC_RTC[5],ALMSrc.ALM_SecondValue) ];
   1: AOI_ALM_Arch(FC_ALM_Arch,FCI_ALMDataLogTrig,ALM_TriggerId,ALMSrc,ALMSer,INTERNAL_RN21_HB_PLC2ServerCommFailed,ALM_UniqueNum,ALMSrc_UniqueNum);
END_ROUTINE

ROUTINE RN21_ALM_Map   (* ladder *)
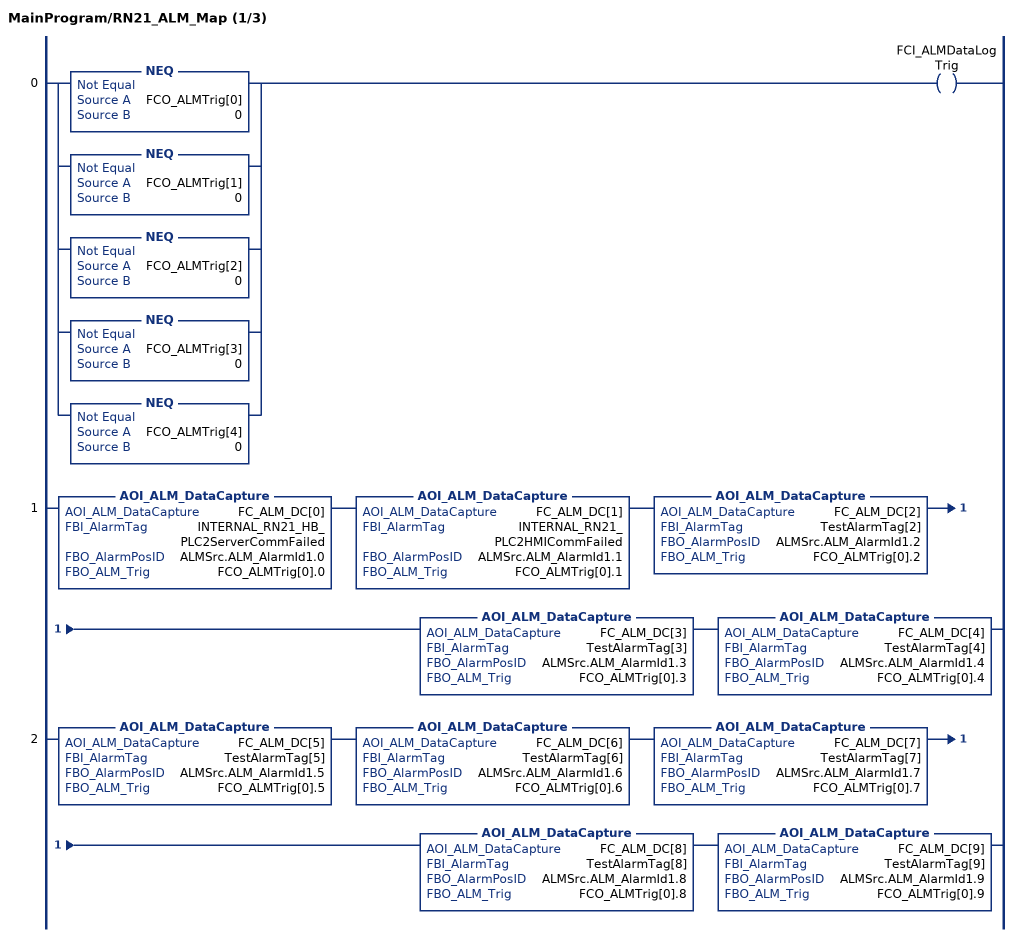
   0: [NEQ(FCO_ALMTrig[0],0) ,NEQ(FCO_ALMTrig[1],0) ,NEQ(FCO_ALMTrig[2],0) ,NEQ(FCO_ALMTrig[3],0) ,NEQ(FCO_ALMTrig[4],0) ]OTE(FCI_ALMDataLogTrig);
   1: AOI_ALM_DataCapture(FC_ALM_DC[0],INTERNAL_RN21_HB_PLC2ServerCommFailed,ALMSrc.ALM_AlarmId1.0,FCO_ALMTrig[0].0)AOI_ALM_DataCapture(FC_ALM_DC[1],INTERNAL_RN21_PLC2HMICommFailed,ALMSrc.ALM_AlarmId1.1,FCO_ALMTrig[0].1)AOI_ALM_DataCapture(FC_ALM_DC[2],TestAlarmTag[2],ALMSrc.ALM_AlarmId1.2,FCO_ALMTrig[0].2)AOI_ALM_DataCapture(FC_ALM_DC[3],TestAlarmTag[3],ALMSrc.ALM_AlarmId1.3,FCO_ALMTrig[0].3)AOI_ALM_DataCapture(FC_ALM_DC[4],TestAlarmTag[4],ALMSrc.ALM_AlarmId1.4,FCO_ALMTrig[0].4);
   2: AOI_ALM_DataCapture(FC_ALM_DC[5],TestAlarmTag[5],ALMSrc.ALM_AlarmId1.5,FCO_ALMTrig[0].5)AOI_ALM_DataCapture(FC_ALM_DC[6],TestAlarmTag[6],ALMSrc.ALM_AlarmId1.6,FCO_ALMTrig[0].6)AOI_ALM_DataCapture(FC_ALM_DC[7],TestAlarmTag[7],ALMSrc.ALM_AlarmId1.7,FCO_ALMTrig[0].7)AOI_ALM_DataCapture(FC_ALM_DC[8],TestAlarmTag[8],ALMSrc.ALM_AlarmId1.8,FCO_ALMTrig[0].8)AOI_ALM_DataCapture(FC_ALM_DC[9],TestAlarmTag[9],ALMSrc.ALM_AlarmId1.9,FCO_ALMTrig[0].9);
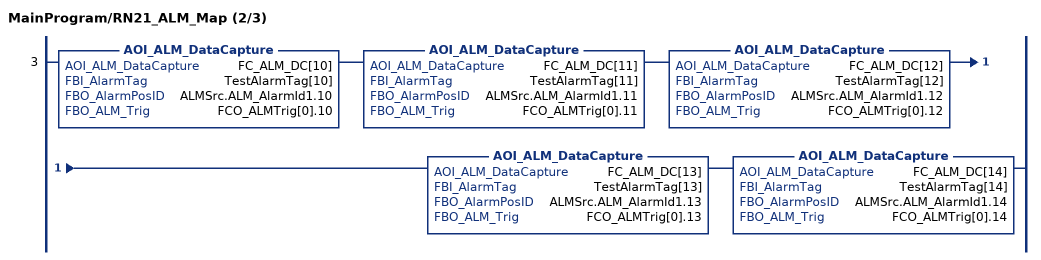
   3: AOI_ALM_DataCapture(FC_ALM_DC[10],TestAlarmTag[10],ALMSrc.ALM_AlarmId1.10,FCO_ALMTrig[0].10)AOI_ALM_DataCapture(FC_ALM_DC[11],TestAlarmTag[11],ALMSrc.ALM_AlarmId1.11,FCO_ALMTrig[0].11)AOI_ALM_DataCapture(FC_ALM_DC[12],TestAlarmTag[12],ALMSrc.ALM_AlarmId1.12,FCO_ALMTrig[0].12)AOI_ALM_DataCapture(FC_ALM_DC[13],TestAlarmTag[13],ALMSrc.ALM_AlarmId1.13,FCO_ALMTrig[0].13)AOI_ALM_DataCapture(FC_ALM_DC[14],TestAlarmTag[14],ALMSrc.ALM_AlarmId1.14,FCO_ALMTrig[0].14);
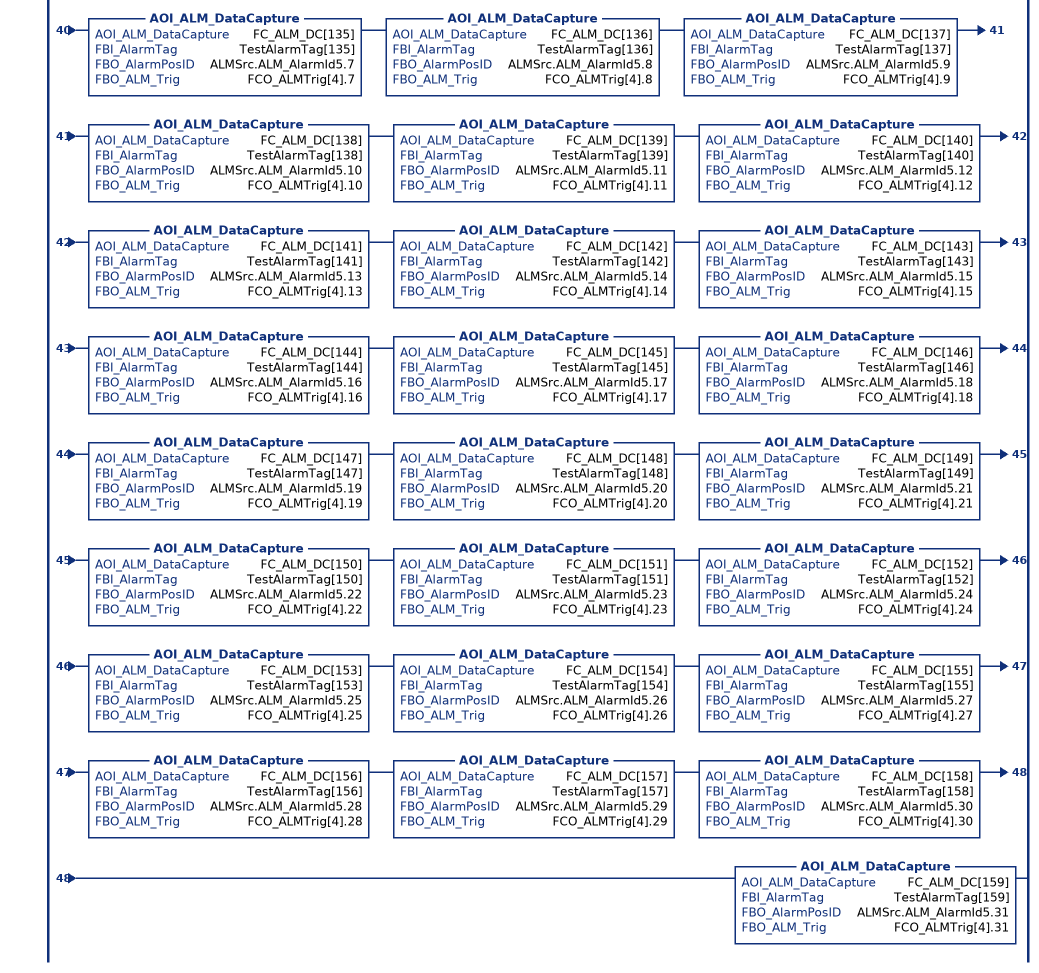
   4: AOI_ALM_DataCapture(FC_ALM_DC[15],TestAlarmTag[15],ALMSrc.ALM_AlarmId1.15,FCO_ALMTrig[0].15)AOI_ALM_DataCapture(FC_ALM_DC[16],TestAlarmTag[16],ALMSrc.ALM_AlarmId1.16,FCO_ALMTrig[0].16)AOI_ALM_DataCapture(FC_ALM_DC[17],TestAlarmTag[17],ALMSrc.ALM_AlarmId1.17,FCO_ALMTrig[0].17)AOI_ALM_DataCapture(FC_ALM_DC[18],TestAlarmTag[18],ALMSrc.ALM_AlarmId1.18,FCO_ALMTrig[0].18)AOI_ALM_DataCapture(FC_ALM_DC[19],TestAlarmTag[19],ALMSrc.ALM_AlarmId1.19,FCO_ALMTrig[0].19)AOI_ALM_DataCapture(FC_ALM_DC[20],TestAlarmTag[20],ALMSrc.ALM_AlarmId1.20,FCO_ALMTrig[0].20)AOI_ALM_DataCapture(FC_ALM_DC[21],TestAlarmTag[21],ALMSrc.ALM_AlarmId1.21,FCO_ALMTrig[0].21)AOI_ALM_DataCapture(FC_ALM_DC[22],TestAlarmTag[22],ALMSrc.ALM_AlarmId1.22,FCO_ALMTrig[0].22)AOI_ALM_DataCapture(FC_ALM_DC[23],TestAlarmTag[23],ALMSrc.ALM_AlarmId1.23,FCO_ALMTrig[0].23)AOI_ALM_DataCapture(FC_ALM_DC[24],TestAlarmTag[24],ALMSrc.ALM_AlarmId1.24,FCO_ALMTrig[0].24)AOI_ALM_DataCapture(FC_ALM_DC[25],TestAlarmTag[25],ALMSrc.ALM_AlarmId1.25,FCO_ALMTrig[0].25)AOI_ALM_DataCapture(FC_ALM_DC[26],TestAlarmTag[26],ALMSrc.ALM_AlarmId1.26,FCO_ALMTrig[0].26)AOI_ALM_DataCapture(FC_ALM_DC[27],TestAlarmTag[27],ALMSrc.ALM_AlarmId1.27,FCO_ALMTrig[0].27)AOI_ALM_DataCapture(FC_ALM_DC[28],TestAlarmTag[28],ALMSrc.ALM_AlarmId1.28,FCO_ALMTrig[0].28)AOI_ALM_DataCapture(FC_ALM_DC[29],TestAlarmTag[29],ALMSrc.ALM_AlarmId1.29,FCO_ALMTrig[0].29)AOI_ALM_DataCapture(FC_ALM_DC[30],TestAlarmTag[30],ALMSrc.ALM_AlarmId1.30,FCO_ALMTrig[0].30)AOI_ALM_DataCapture(FC_ALM_DC[31],TestAlarmTag[31],ALMSrc.ALM_AlarmId1.31,FCO_ALMTrig[0].31)AOI_ALM_DataCapture(FC_ALM_DC[32],TestAlarmTag[32],ALMSrc.ALM_AlarmId2.0,FCO_ALMTrig[1].0)AOI_ALM_DataCapture(FC_ALM_DC[33],TestAlarmTag[33],ALMSrc.ALM_AlarmId2.1,FCO_ALMTrig[1].1)AOI_ALM_DataCapture(FC_ALM_DC[34],TestAlarmTag[34],ALMSrc.ALM_AlarmId2.2,FCO_ALMTrig[1].2)AOI_ALM_DataCapture(FC_ALM_DC[35],TestAlarmTag[35],ALMSrc.ALM_AlarmId2.3,FCO_ALMTrig[1].3)AOI_ALM_DataCapture(FC_ALM_DC[36],TestAlarmTag[36],ALMSrc.ALM_AlarmId2.4,FCO_ALMTrig[1].4)AOI_ALM_DataCapture(FC_ALM_DC[37],TestAlarmTag[37],ALMSrc.ALM_AlarmId2.5,FCO_ALMTrig[1].5)AOI_ALM_DataCapture(FC_ALM_DC[38],TestAlarmTag[38],ALMSrc.ALM_AlarmId2.6,FCO_ALMTrig[1].6)AOI_ALM_DataCapture(FC_ALM_DC[39],TestAlarmTag[39],ALMSrc.ALM_AlarmId2.7,FCO_ALMTrig[1].7)AOI_ALM_DataCapture(FC_ALM_DC[40],TestAlarmTag[40],ALMSrc.ALM_AlarmId2.8,FCO_ALMTrig[1].8)AOI_ALM_DataCapture(FC_ALM_DC[41],TestAlarmTag[41],ALMSrc.ALM_AlarmId2.9,FCO_ALMTrig[1].9)AOI_ALM_DataCapture(FC_ALM_DC[42],TestAlarmTag[42],ALMSrc.ALM_AlarmId2.10,FCO_ALMTrig[1].10)AOI_ALM_DataCapture(FC_ALM_DC[43],TestAlarmTag[43],ALMSrc.ALM_AlarmId2.11,FCO_ALMTrig[1].11)AOI_ALM_DataCapture(FC_ALM_DC[44],TestAlarmTag[44],ALMSrc.ALM_AlarmId2.12,FCO_ALMTrig[1].12)AOI_ALM_DataCapture(FC_ALM_DC[45],TestAlarmTag[45],ALMSrc.ALM_AlarmId2.13,FCO_ALMTrig[1].13)AOI_ALM_DataCapture(FC_ALM_DC[46],TestAlarmTag[46],ALMSrc.ALM_AlarmId2.14,FCO_ALMTrig[1].14)AOI_ALM_DataCapture(FC_ALM_DC[47],TestAlarmTag[47],ALMSrc.ALM_AlarmId2.15,FCO_ALMTrig[1].15)AOI_ALM_DataCapture(FC_ALM_DC[48],TestAlarmTag[48],ALMSrc.ALM_AlarmId2.16,FCO_ALMTrig[1].16)AOI_ALM_DataCapture(FC_ALM_DC[49],TestAlarmTag[49],ALMSrc.ALM_AlarmId2.17,FCO_ALMTrig[1].17)AOI_ALM_DataCapture(FC_ALM_DC[50],TestAlarmTag[50],ALMSrc.ALM_AlarmId2.18,FCO_ALMTrig[1].18)AOI_ALM_DataCapture(FC_ALM_DC[51],TestAlarmTag[51],ALMSrc.ALM_AlarmId2.19,FCO_ALMTrig[1].19)AOI_ALM_DataCapture(FC_ALM_DC[52],TestAlarmTag[52],ALMSrc.ALM_AlarmId2.20,FCO_ALMTrig[1].20)AOI_ALM_DataCapture(FC_ALM_DC[53],TestAlarmTag[53],ALMSrc.ALM_AlarmId2.21,FCO_ALMTrig[1].21)AOI_ALM_DataCapture(FC_ALM_DC[54],TestAlarmTag[54],ALMSrc.ALM_AlarmId2.22,FCO_ALMTrig[1].22)AOI_ALM_DataCapture(FC_ALM_DC[55],TestAlarmTag[55],ALMSrc.ALM_AlarmId2.23,FCO_ALMTrig[1].23)AOI_ALM_DataCapture(FC_ALM_DC[56],TestAlarmTag[56],ALMSrc.ALM_AlarmId2.24,FCO_ALMTrig[1].24)AOI_ALM_DataCapture(FC_ALM_DC[57],TestAlarmTag[57],ALMSrc.ALM_AlarmId2.25,FCO_ALMTrig[1].25)AOI_ALM_DataCapture(FC_ALM_DC[58],TestAlarmTag[58],ALMSrc.ALM_AlarmId2.26,FCO_ALMTrig[1].26)AOI_ALM_DataCapture(FC_ALM_DC[59],TestAlarmTag[59],ALMSrc.ALM_AlarmId2.27,FCO_ALMTrig[1].27)AOI_ALM_DataCapture(FC_ALM_DC[60],TestAlarmTag[60],ALMSrc.ALM_AlarmId2.28,FCO_ALMTrig[1].28)AOI_ALM_DataCapture(FC_ALM_DC[61],TestAlarmTag[61],ALMSrc.ALM_AlarmId2.29,FCO_ALMTrig[1].29)AOI_ALM_DataCapture(FC_ALM_DC[62],TestAlarmTag[62],ALMSrc.ALM_AlarmId2.30,FCO_ALMTrig[1].30)AOI_ALM_DataCapture(FC_ALM_DC[63],TestAlarmTag[63],ALMSrc.ALM_AlarmId2.31,FCO_ALMTrig[1].31)AOI_ALM_DataCapture(FC_ALM_DC[64],TestAlarmTag[64],ALMSrc.ALM_AlarmId3.0,FCO_ALMTrig[2].0)AOI_ALM_DataCapture(FC_ALM_DC[65],TestAlarmTag[65],ALMSrc.ALM_AlarmId3.1,FCO_ALMTrig[2].1)AOI_ALM_DataCapture(FC_ALM_DC[66],TestAlarmTag[66],ALMSrc.ALM_AlarmId3.2,FCO_ALMTrig[2].2)AOI_ALM_DataCapture(FC_ALM_DC[67],TestAlarmTag[67],ALMSrc.ALM_AlarmId3.3,FCO_ALMTrig[2].3)AOI_ALM_DataCapture(FC_ALM_DC[68],TestAlarmTag[68],ALMSrc.ALM_AlarmId3.4,FCO_ALMTrig[2].4)AOI_ALM_DataCapture(FC_ALM_DC[69],TestAlarmTag[69],ALMSrc.ALM_AlarmId3.5,FCO_ALMTrig[2].5)AOI_ALM_DataCapture(FC_ALM_DC[70],TestAlarmTag[70],ALMSrc.ALM_AlarmId3.6,FCO_ALMTrig[2].6)AOI_ALM_DataCapture(FC_ALM_DC[71],TestAlarmTag[71],ALMSrc.ALM_AlarmId3.7,FCO_ALMTrig[2].7)AOI_ALM_DataCapture(FC_ALM_DC[72],TestAlarmTag[72],ALMSrc.ALM_AlarmId3.8,FCO_ALMTrig[2].8)AOI_ALM_DataCapture(FC_ALM_DC[73],TestAlarmTag[73],ALMSrc.ALM_AlarmId3.9,FCO_ALMTrig[2].9)AOI_ALM_DataCapture(FC_ALM_DC[74],TestAlarmTag[74],ALMSrc.ALM_AlarmId3.10,FCO_ALMTrig[2].10)AOI_ALM_DataCapture(FC_ALM_DC[75],TestAlarmTag[75],ALMSrc.ALM_AlarmId3.11,FCO_ALMTrig[2].11)AOI_ALM_DataCapture(FC_ALM_DC[76],TestAlarmTag[76],ALMSrc.ALM_AlarmId3.12,FCO_ALMTrig[2].12)AOI_ALM_DataCapture(FC_ALM_DC[77],TestAlarmTag[77],ALMSrc.ALM_AlarmId3.13,FCO_ALMTrig[2].13)AOI_ALM_DataCapture(FC_ALM_DC[78],TestAlarmTag[78],ALMSrc.ALM_AlarmId3.14,FCO_ALMTrig[2].14)AOI_ALM_DataCapture(FC_ALM_DC[79],TestAlarmTag[79],ALMSrc.ALM_AlarmId3.15,FCO_ALMTrig[2].15)AOI_ALM_DataCapture(FC_ALM_DC[80],TestAlarmTag[80],ALMSrc.ALM_AlarmId3.16,FCO_ALMTrig[2].16)AOI_ALM_DataCapture(FC_ALM_DC[81],TestAlarmTag[81],ALMSrc.ALM_AlarmId3.17,FCO_ALMTrig[2].17)AOI_ALM_DataCapture(FC_ALM_DC[82],TestAlarmTag[82],ALMSrc.ALM_AlarmId3.18,FCO_ALMTrig[2].18)AOI_ALM_DataCapture(FC_ALM_DC[83],TestAlarmTag[83],ALMSrc.ALM_AlarmId3.19,FCO_ALMTrig[2].19)AOI_ALM_DataCapture(FC_ALM_DC[84],TestAlarmTag[84],ALMSrc.ALM_AlarmId3.20,FCO_ALMTrig[2].20)AOI_ALM_DataCapture(FC_ALM_DC[85],TestAlarmTag[85],ALMSrc.ALM_AlarmId3.21,FCO_ALMTrig[2].21)AOI_ALM_DataCapture(FC_ALM_DC[86],TestAlarmTag[86],ALMSrc.ALM_AlarmId3.22,FCO_ALMTrig[2].22)AOI_ALM_DataCapture(FC_ALM_DC[87],TestAlarmTag[87],ALMSrc.ALM_AlarmId3.23,FCO_ALMTrig[2].23)AOI_ALM_DataCapture(FC_ALM_DC[88],TestAlarmTag[88],ALMSrc.ALM_AlarmId3.24,FCO_ALMTrig[2].24)AOI_ALM_DataCapture(FC_ALM_DC[89],TestAlarmTag[89],ALMSrc.ALM_AlarmId3.25,FCO_ALMTrig[2].25)AOI_ALM_DataCapture(FC_ALM_DC[90],TestAlarmTag[90],ALMSrc.ALM_AlarmId3.26,FCO_ALMTrig[2].26)AOI_ALM_DataCapture(FC_ALM_DC[91],TestAlarmTag[91],ALMSrc.ALM_AlarmId3.27,FCO_ALMTrig[2].27)AOI_ALM_DataCapture(FC_ALM_DC[92],TestAlarmTag[92],ALMSrc.ALM_AlarmId3.28,FCO_ALMTrig[2].28)AOI_ALM_DataCapture(FC_ALM_DC[93],TestAlarmTag[93],ALMSrc.ALM_AlarmId3.29,FCO_ALMTrig[2].29)AOI_ALM_DataCapture(FC_ALM_DC[94],TestAlarmTag[94],ALMSrc.ALM_AlarmId3.30,FCO_ALMTrig[2].30)AOI_ALM_DataCapture(FC_ALM_DC[95],TestAlarmTag[95],ALMSrc.ALM_AlarmId3.31,FCO_ALMTrig[2].31)AOI_ALM_DataCapture(FC_ALM_DC[96],TestAlarmTag[96],ALMSrc.ALM_AlarmId4.0,FCO_ALMTrig[3].0)AOI_ALM_DataCapture(FC_ALM_DC[97],TestAlarmTag[97],ALMSrc.ALM_AlarmId4.1,FCO_ALMTrig[3].1)AOI_ALM_DataCapture(FC_ALM_DC[98],TestAlarmTag[98],ALMSrc.ALM_AlarmId4.2,FCO_ALMTrig[3].2)AOI_ALM_DataCapture(FC_ALM_DC[99],TestAlarmTag[99],ALMSrc.ALM_AlarmId4.3,FCO_ALMTrig[3].3)AOI_ALM_DataCapture(FC_ALM_DC[100],TestAlarmTag[100],ALMSrc.ALM_AlarmId4.4,FCO_ALMTrig[3].4)AOI_ALM_DataCapture(FC_ALM_DC[101],TestAlarmTag[101],ALMSrc.ALM_AlarmId4.5,FCO_ALMTrig[3].5)AOI_ALM_DataCapture(FC_ALM_DC[102],TestAlarmTag[102],ALMSrc.ALM_AlarmId4.6,FCO_ALMTrig[3].6)AOI_ALM_DataCapture(FC_ALM_DC[103],TestAlarmTag[103],ALMSrc.ALM_AlarmId4.7,FCO_ALMTrig[3].7)AOI_ALM_DataCapture(FC_ALM_DC[104],TestAlarmTag[104],ALMSrc.ALM_AlarmId4.8,FCO_ALMTrig[3].8)AOI_ALM_DataCapture(FC_ALM_DC[105],TestAlarmTag[105],ALMSrc.ALM_AlarmId4.9,FCO_ALMTrig[3].9)AOI_ALM_DataCapture(FC_ALM_DC[106],TestAlarmTag[106],ALMSrc.ALM_AlarmId4.10,FCO_ALMTrig[3].10)AOI_ALM_DataCapture(FC_ALM_DC[107],TestAlarmTag[107],ALMSrc.ALM_AlarmId4.11,FCO_ALMTrig[3].11)AOI_ALM_DataCapture(FC_ALM_DC[108],TestAlarmTag[108],ALMSrc.ALM_AlarmId4.12,FCO_ALMTrig[3].12)AOI_ALM_DataCapture(FC_ALM_DC[109],TestAlarmTag[109],ALMSrc.ALM_AlarmId4.13,FCO_ALMTrig[3].13)AOI_ALM_DataCapture(FC_ALM_DC[110],TestAlarmTag[110],ALMSrc.ALM_AlarmId4.14,FCO_ALMTrig[3].14)AOI_ALM_DataCapture(FC_ALM_DC[111],TestAlarmTag[111],ALMSrc.ALM_AlarmId4.15,FCO_ALMTrig[3].15)AOI_ALM_DataCapture(FC_ALM_DC[112],TestAlarmTag[112],ALMSrc.ALM_AlarmId4.16,FCO_ALMTrig[3].16)AOI_ALM_DataCapture(FC_ALM_DC[113],TestAlarmTag[113],ALMSrc.ALM_AlarmId4.17,FCO_ALMTrig[3].17)AOI_ALM_DataCapture(FC_ALM_DC[114],TestAlarmTag[114],ALMSrc.ALM_AlarmId4.18,FCO_ALMTrig[3].18)AOI_ALM_DataCapture(FC_ALM_DC[115],TestAlarmTag[115],ALMSrc.ALM_AlarmId4.19,FCO_ALMTrig[3].19)AOI_ALM_DataCapture(FC_ALM_DC[116],TestAlarmTag[116],ALMSrc.ALM_AlarmId4.20,FCO_ALMTrig[3].20)AOI_ALM_DataCapture(FC_ALM_DC[117],TestAlarmTag[117],ALMSrc.ALM_AlarmId4.21,FCO_ALMTrig[3].21)AOI_ALM_DataCapture(FC_ALM_DC[118],TestAlarmTag[118],ALMSrc.ALM_AlarmId4.22,FCO_ALMTrig[3].22)AOI_ALM_DataCapture(FC_ALM_DC[119],TestAlarmTag[119],ALMSrc.ALM_AlarmId4.23,FCO_ALMTrig[3].23)AOI_ALM_DataCapture(FC_ALM_DC[120],TestAlarmTag[120],ALMSrc.ALM_AlarmId4.24,FCO_ALMTrig[3].24)AOI_ALM_DataCapture(FC_ALM_DC[121],TestAlarmTag[121],ALMSrc.ALM_AlarmId4.25,FCO_ALMTrig[3].25)AOI_ALM_DataCapture(FC_ALM_DC[122],TestAlarmTag[122],ALMSrc.ALM_AlarmId4.26,FCO_ALMTrig[3].26)AOI_ALM_DataCapture(FC_ALM_DC[123],TestAlarmTag[123],ALMSrc.ALM_AlarmId4.27,FCO_ALMTrig[3].27)AOI_ALM_DataCapture(FC_ALM_DC[124],TestAlarmTag[124],ALMSrc.ALM_AlarmId4.28,FCO_ALMTrig[3].28)AOI_ALM_DataCapture(FC_ALM_DC[125],TestAlarmTag[125],ALMSrc.ALM_AlarmId4.29,FCO_ALMTrig[3].29)AOI_ALM_DataCapture(FC_ALM_DC[126],TestAlarmTag[126],ALMSrc.ALM_AlarmId4.30,FCO_ALMTrig[3].30)AOI_ALM_DataCapture(FC_ALM_DC[127],TestAlarmTag[127],ALMSrc.ALM_AlarmId4.31,FCO_ALMTrig[3].31)AOI_ALM_DataCapture(FC_ALM_DC[128],TestAlarmTag[128],ALMSrc.ALM_AlarmId5.0,FCO_ALMTrig[4].0)AOI_ALM_DataCapture(FC_ALM_DC[129],TestAlarmTag[129],ALMSrc.ALM_AlarmId5.1,FCO_ALMTrig[4].1)AOI_ALM_DataCapture(FC_ALM_DC[130],TestAlarmTag[130],ALMSrc.ALM_AlarmId5.2,FCO_ALMTrig[4].2)AOI_ALM_DataCapture(FC_ALM_DC[131],TestAlarmTag[131],ALMSrc.ALM_AlarmId5.3,FCO_ALMTrig[4].3)AOI_ALM_DataCapture(FC_ALM_DC[132],TestAlarmTag[132],ALMSrc.ALM_AlarmId5.4,FCO_ALMTrig[4].4)AOI_ALM_DataCapture(FC_ALM_DC[133],TestAlarmTag[133],ALMSrc.ALM_AlarmId5.5,FCO_ALMTrig[4].5)AOI_ALM_DataCapture(FC_ALM_DC[134],TestAlarmTag[134],ALMSrc.ALM_AlarmId5.6,FCO_ALMTrig[4].6)AOI_ALM_DataCapture(FC_ALM_DC[135],TestAlarmTag[135],ALMSrc.ALM_AlarmId5.7,FCO_ALMTrig[4].7)AOI_ALM_DataCapture(FC_ALM_DC[136],TestAlarmTag[136],ALMSrc.ALM_AlarmId5.8,FCO_ALMTrig[4].8)AOI_ALM_DataCapture(FC_ALM_DC[137],TestAlarmTag[137],ALMSrc.ALM_AlarmId5.9,FCO_ALMTrig[4].9)AOI_ALM_DataCapture(FC_ALM_DC[138],TestAlarmTag[138],ALMSrc.ALM_AlarmId5.10,FCO_ALMTrig[4].10)AOI_ALM_DataCapture(FC_ALM_DC[139],TestAlarmTag[139],ALMSrc.ALM_AlarmId5.11,FCO_ALMTrig[4].11)AOI_ALM_DataCapture(FC_ALM_DC[140],TestAlarmTag[140],ALMSrc.ALM_AlarmId5.12,FCO_ALMTrig[4].12)AOI_ALM_DataCapture(FC_ALM_DC[141],TestAlarmTag[141],ALMSrc.ALM_AlarmId5.13,FCO_ALMTrig[4].13)AOI_ALM_DataCapture(FC_ALM_DC[142],TestAlarmTag[142],ALMSrc.ALM_AlarmId5.14,FCO_ALMTrig[4].14)AOI_ALM_DataCapture(FC_ALM_DC[143],TestAlarmTag[143],ALMSrc.ALM_AlarmId5.15,FCO_ALMTrig[4].15)AOI_ALM_DataCapture(FC_ALM_DC[144],TestAlarmTag[144],ALMSrc.ALM_AlarmId5.16,FCO_ALMTrig[4].16)AOI_ALM_DataCapture(FC_ALM_DC[145],TestAlarmTag[145],ALMSrc.ALM_AlarmId5.17,FCO_ALMTrig[4].17)AOI_ALM_DataCapture(FC_ALM_DC[146],TestAlarmTag[146],ALMSrc.ALM_AlarmId5.18,FCO_ALMTrig[4].18)AOI_ALM_DataCapture(FC_ALM_DC[147],TestAlarmTag[147],ALMSrc.ALM_AlarmId5.19,FCO_ALMTrig[4].19)AOI_ALM_DataCapture(FC_ALM_DC[148],TestAlarmTag[148],ALMSrc.ALM_AlarmId5.20,FCO_ALMTrig[4].20)AOI_ALM_DataCapture(FC_ALM_DC[149],TestAlarmTag[149],ALMSrc.ALM_AlarmId5.21,FCO_ALMTrig[4].21)AOI_ALM_DataCapture(FC_ALM_DC[150],TestAlarmTag[150],ALMSrc.ALM_AlarmId5.22,FCO_ALMTrig[4].22)AOI_ALM_DataCapture(FC_ALM_DC[151],TestAlarmTag[151],ALMSrc.ALM_AlarmId5.23,FCO_ALMTrig[4].23)AOI_ALM_DataCapture(FC_ALM_DC[152],TestAlarmTag[152],ALMSrc.ALM_AlarmId5.24,FCO_ALMTrig[4].24)AOI_ALM_DataCapture(FC_ALM_DC[153],TestAlarmTag[153],ALMSrc.ALM_AlarmId5.25,FCO_ALMTrig[4].25)AOI_ALM_DataCapture(FC_ALM_DC[154],TestAlarmTag[154],ALMSrc.ALM_AlarmId5.26,FCO_ALMTrig[4].26)AOI_ALM_DataCapture(FC_ALM_DC[155],TestAlarmTag[155],ALMSrc.ALM_AlarmId5.27,FCO_ALMTrig[4].27)AOI_ALM_DataCapture(FC_ALM_DC[156],TestAlarmTag[156],ALMSrc.ALM_AlarmId5.28,FCO_ALMTrig[4].28)AOI_ALM_DataCapture(FC_ALM_DC[157],TestAlarmTag[157],ALMSrc.ALM_AlarmId5.29,FCO_ALMTrig[4].29)AOI_ALM_DataCapture(FC_ALM_DC[158],TestAlarmTag[158],ALMSrc.ALM_AlarmId5.30,FCO_ALMTrig[4].30)AOI_ALM_DataCapture(FC_ALM_DC[159],TestAlarmTag[159],ALMSrc.ALM_AlarmId5.31,FCO_ALMTrig[4].31);
END_ROUTINE

ROUTINE RN21_AUD_Main   (* ladder *)
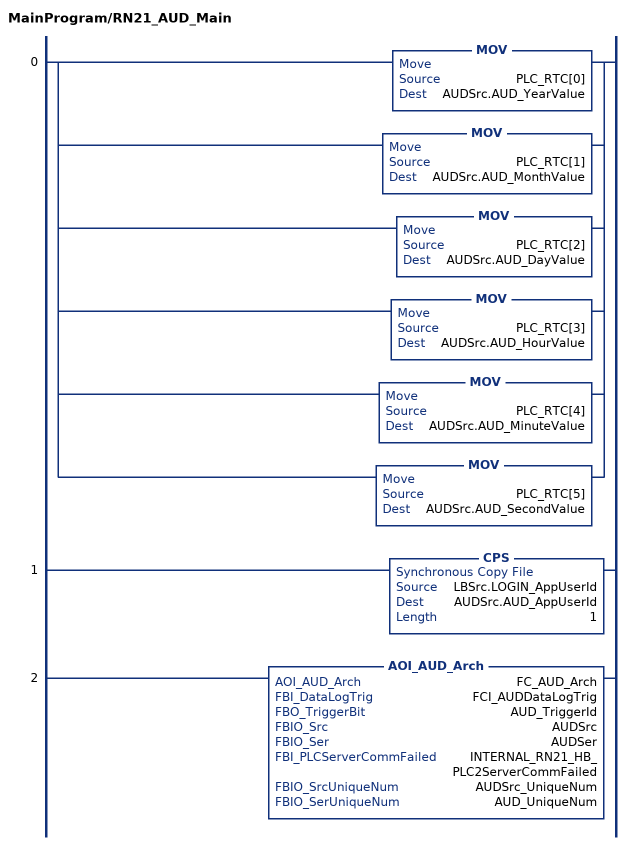
   0: [MOV(PLC_RTC[0],AUDSrc.AUD_YearValue) ,MOV(PLC_RTC[1],AUDSrc.AUD_MonthValue) ,MOV(PLC_RTC[2],AUDSrc.AUD_DayValue) ,MOV(PLC_RTC[3],AUDSrc.AUD_HourValue) ,MOV(PLC_RTC[4],AUDSrc.AUD_MinuteValue) ,MOV(PLC_RTC[5],AUDSrc.AUD_SecondValue) ];
   1: CPS(LBSrc.LOGIN_AppUserId,AUDSrc.AUD_AppUserId,1);
   2: AOI_AUD_Arch(FC_AUD_Arch,FCI_AUDDataLogTrig,AUD_TriggerId,AUDSrc,AUDSer,INTERNAL_RN21_HB_PLC2ServerCommFailed,AUDSrc_UniqueNum,AUD_UniqueNum);
END_ROUTINE

ROUTINE RN21_AUD_Map   (* ladder *)
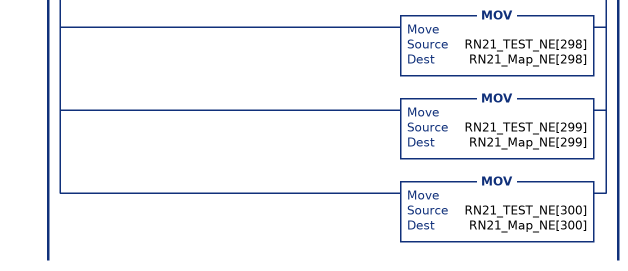
   // Numeric Entry Mapping
   0: [MOV(RN21_TEST_NE[0],RN21_Map_NE[0]) ,MOV(RN21_TEST_NE[1],RN21_Map_NE[1]) ,MOV(RN21_TEST_NE[2],RN21_Map_NE[2]) ,MOV(RN21_TEST_NE[3],RN21_Map_NE[3]) ,MOV(RN21_TEST_NE[4],RN21_Map_NE[4]) ,MOV(RN21_TEST_NE[5],RN21_Map_NE[5]) ,MOV(RN21_TEST_NE[6],RN21_Map_NE[6]) ,MOV(RN21_TEST_NE[7],RN21_Map_NE[7]) ,MOV(RN21_TEST_NE[8],RN21_Map_NE[8]) ,MOV(RN21_TEST_NE[9],RN21_Map_NE[9]) ,MOV(RN21_TEST_NE[10],RN21_Map_NE[10]) ,MOV(RN21_TEST_NE[11],RN21_Map_NE[11]) ,MOV(RN21_TEST_NE[12],RN21_Map_NE[12]) ,MOV(RN21_TEST_NE[13],RN21_Map_NE[13]) ,MOV(RN21_TEST_NE[14],RN21_Map_NE[14]) ,MOV(RN21_TEST_NE[15],RN21_Map_NE[15]) ,MOV(RN21_TEST_NE[16],RN21_Map_NE[16]) ,MOV(RN21_TEST_NE[17],RN21_Map_NE[17]) ,MOV(RN21_TEST_NE[18],RN21_Map_NE[18]) ,MOV(RN21_TEST_NE[19],RN21_Map_NE[19]) ,MOV(RN21_TEST_NE[20],RN21_Map_NE[20]) ,MOV(RN21_TEST_NE[21],RN21_Map_NE[21]) ,MOV(RN21_TEST_NE[22],RN21_Map_NE[22]) ,MOV(RN21_TEST_NE[23],RN21_Map_NE[23]) ,MOV(RN21_TEST_NE[24],RN21_Map_NE[24]) ,MOV(RN21_TEST_NE[25],RN21_Map_NE[25]) ,MOV(RN21_TEST_NE[26],RN21_Map_NE[26]) ,MOV(RN21_TEST_NE[27],RN21_Map_NE[27]) ,MOV(RN21_TEST_NE[28],RN21_Map_NE[28]) ,MOV(RN21_TEST_NE[29],RN21_Map_NE[29]) ,MOV(RN21_TEST_NE[30],RN21_Map_NE[30]) ,MOV(RN21_TEST_NE[31],RN21_Map_NE[31]) ,MOV(RN21_TEST_NE[32],RN21_Map_NE[32]) ,MOV(RN21_TEST_NE[33],RN21_Map_NE[33]) ,MOV(RN21_TEST_NE[34],RN21_Map_NE[34]) ,MOV(RN21_TEST_NE[35],RN21_Map_NE[35]) ,MOV(RN21_TEST_NE[36],RN21_Map_NE[36]) ,MOV(RN21_TEST_NE[37],RN21_Map_NE[37]) ,MOV(RN21_TEST_NE[38],RN21_Map_NE[38]) ,MOV(RN21_TEST_NE[39],RN21_Map_NE[39]) ,MOV(RN21_TEST_NE[40],RN21_Map_NE[40]) ,MOV(RN21_TEST_NE[41],RN21_Map_NE[41]) ,MOV(RN21_TEST_NE[42],RN21_Map_NE[42]) ,MOV(RN21_TEST_NE[43],RN21_Map_NE[43]) ,MOV(RN21_TEST_NE[44],RN21_Map_NE[44]) ,MOV(RN21_TEST_NE[45],RN21_Map_NE[45]) ,MOV(RN21_TEST_NE[46],RN21_Map_NE[46]) ,MOV(RN21_TEST_NE[47],RN21_Map_NE[47]) ,MOV(RN21_TEST_NE[48],RN21_Map_NE[48]) ,MOV(RN21_TEST_NE[49],RN21_Map_NE[49]) ,MOV(RN21_TEST_NE[50],RN21_Map_NE[50]) ,MOV(RN21_TEST_NE[51],RN21_Map_NE[51]) ,MOV(RN21_TEST_NE[52],RN21_Map_NE[52]) ,MOV(RN21_TEST_NE[53],RN21_Map_NE[53]) ,MOV(RN21_TEST_NE[54],RN21_Map_NE[54]) ,MOV(RN21_TEST_NE[55],RN21_Map_NE[55]) ,MOV(RN21_TEST_NE[56],RN21_Map_NE[56]) ,MOV(RN21_TEST_NE[57],RN21_Map_NE[57]) ,MOV(RN21_TEST_NE[58],RN21_Map_NE[58]) ,MOV(RN21_TEST_NE[59],RN21_Map_NE[59]) ,MOV(RN21_TEST_NE[60],RN21_Map_NE[60]) ,MOV(RN21_TEST_NE[61],RN21_Map_NE[61]) ,MOV(RN21_TEST_NE[62],RN21_Map_NE[62]) ,MOV(RN21_TEST_NE[63],RN21_Map_NE[63]) ,MOV(RN21_TEST_NE[64],RN21_Map_NE[64]) ,MOV(RN21_TEST_NE[65],RN21_Map_NE[65]) ,MOV(RN21_TEST_NE[66],RN21_Map_NE[66]) ,MOV(RN21_TEST_NE[67],RN21_Map_NE[67]) ,MOV(RN21_TEST_NE[68],RN21_Map_NE[68]) ,MOV(RN21_TEST_NE[69],RN21_Map_NE[69]) ,MOV(RN21_TEST_NE[70],RN21_Map_NE[70]) ,MOV(RN21_TEST_NE[71],RN21_Map_NE[71]) ,MOV(RN21_TEST_NE[72],RN21_Map_NE[72]) ,MOV(RN21_TEST_NE[73],RN21_Map_NE[73]) ,MOV(RN21_TEST_NE[74],RN21_Map_NE[74]) ,MOV(RN21_TEST_NE[75],RN21_Map_NE[75]) ,MOV(RN21_TEST_NE[76],RN21_Map_NE[76]) ,MOV(RN21_TEST_NE[77],RN21_Map_NE[77]) ,MOV(RN21_TEST_NE[78],RN21_Map_NE[78]) ,MOV(RN21_TEST_NE[79],RN21_Map_NE[79]) ,MOV(RN21_TEST_NE[80],RN21_Map_NE[80]) ,MOV(RN21_TEST_NE[81],RN21_Map_NE[81]) ,MOV(RN21_TEST_NE[82],RN21_Map_NE[82]) ,MOV(RN21_TEST_NE[83],RN21_Map_NE[83]) ,MOV(RN21_TEST_NE[84],RN21_Map_NE[84]) ,MOV(RN21_TEST_NE[85],RN21_Map_NE[85]) ,MOV(RN21_TEST_NE[86],RN21_Map_NE[86]) ,MOV(RN21_TEST_NE[87],RN21_Map_NE[87]) ,MOV(RN21_TEST_NE[88],RN21_Map_NE[88]) ,MOV(RN21_TEST_NE[89],RN21_Map_NE[89]) ,MOV(RN21_TEST_NE[90],RN21_Map_NE[90]) ,MOV(RN21_TEST_NE[91],RN21_Map_NE[91]) ,MOV(RN21_TEST_NE[92],RN21_Map_NE[92]) ,MOV(RN21_TEST_NE[93],RN21_Map_NE[93]) ,MOV(RN21_TEST_NE[94],RN21_Map_NE[94]) ,MOV(RN21_TEST_NE[95],RN21_Map_NE[95]) ,MOV(RN21_TEST_NE[96],RN21_Map_NE[96]) ,MOV(RN21_TEST_NE[97],RN21_Map_NE[97]) ,MOV(RN21_TEST_NE[98],RN21_Map_NE[98]) ,MOV(RN21_TEST_NE[99],RN21_Map_NE[99]) ,MOV(RN21_TEST_NE[100],RN21_Map_NE[100]) ,MOV(RN21_TEST_NE[101],RN21_Map_NE[101]) ,MOV(RN21_TEST_NE[102],RN21_Map_NE[102]) ,MOV(RN21_TEST_NE[103],RN21_Map_NE[103]) ,MOV(RN21_TEST_NE[104],RN21_Map_NE[104]) ,MOV(RN21_TEST_NE[105],RN21_Map_NE[105]) ,MOV(RN21_TEST_NE[106],RN21_Map_NE[106]) ,MOV(RN21_TEST_NE[107],RN21_Map_NE[107]) ,MOV(RN21_TEST_NE[108],RN21_Map_NE[108]) ,MOV(RN21_TEST_NE[109],RN21_Map_NE[109]) ,MOV(RN21_TEST_NE[110],RN21_Map_NE[110]) ,MOV(RN21_TEST_NE[111],RN21_Map_NE[111]) ,MOV(RN21_TEST_NE[112],RN21_Map_NE[112]) ,MOV(RN21_TEST_NE[113],RN21_Map_NE[113]) ,MOV(RN21_TEST_NE[114],RN21_Map_NE[114]) ,MOV(RN21_TEST_NE[115],RN21_Map_NE[115]) ,MOV(RN21_TEST_NE[116],RN21_Map_NE[116]) ,MOV(RN21_TEST_NE[117],RN21_Map_NE[117]) ,MOV(RN21_TEST_NE[118],RN21_Map_NE[118]) ,MOV(RN21_TEST_NE[119],RN21_Map_NE[119]) ,MOV(RN21_TEST_NE[120],RN21_Map_NE[120]) ,MOV(RN21_TEST_NE[121],RN21_Map_NE[121]) ,MOV(RN21_TEST_NE[122],RN21_Map_NE[122]) ,MOV(RN21_TEST_NE[123],RN21_Map_NE[123]) ,MOV(RN21_TEST_NE[124],RN21_Map_NE[124]) ,MOV(RN21_TEST_NE[125],RN21_Map_NE[125]) ,MOV(RN21_TEST_NE[126],RN21_Map_NE[126]) ,MOV(RN21_TEST_NE[127],RN21_Map_NE[127]) ,MOV(RN21_TEST_NE[128],RN21_Map_NE[128]) ,MOV(RN21_TEST_NE[129],RN21_Map_NE[129]) ,MOV(RN21_TEST_NE[130],RN21_Map_NE[130]) ,MOV(RN21_TEST_NE[131],RN21_Map_NE[131]) ,MOV(RN21_TEST_NE[132],RN21_Map_NE[132]) ,MOV(RN21_TEST_NE[133],RN21_Map_NE[133]) ,MOV(RN21_TEST_NE[134],RN21_Map_NE[134]) ,MOV(RN21_TEST_NE[135],RN21_Map_NE[135]) ,MOV(RN21_TEST_NE[136],RN21_Map_NE[136]) ,MOV(RN21_TEST_NE[137],RN21_Map_NE[137]) ,MOV(RN21_TEST_NE[138],RN21_Map_NE[138]) ,MOV(RN21_TEST_NE[139],RN21_Map_NE[139]) ,MOV(RN21_TEST_NE[140],RN21_Map_NE[140]) ,MOV(RN21_TEST_NE[141],RN21_Map_NE[141]) ,MOV(RN21_TEST_NE[142],RN21_Map_NE[142]) ,MOV(RN21_TEST_NE[143],RN21_Map_NE[143]) ,MOV(RN21_TEST_NE[144],RN21_Map_NE[144]) ,MOV(RN21_TEST_NE[145],RN21_Map_NE[145]) ,MOV(RN21_TEST_NE[146],RN21_Map_NE[146]) ,MOV(RN21_TEST_NE[147],RN21_Map_NE[147]) ,MOV(RN21_TEST_NE[148],RN21_Map_NE[148]) ,MOV(RN21_TEST_NE[149],RN21_Map_NE[149]) ,MOV(RN21_TEST_NE[150],RN21_Map_NE[150]) ,MOV(RN21_TEST_NE[151],RN21_Map_NE[151]) ,MOV(RN21_TEST_NE[152],RN21_Map_NE[152]) ,MOV(RN21_TEST_NE[153],RN21_Map_NE[153]) ,MOV(RN21_TEST_NE[154],RN21_Map_NE[154]) ,MOV(RN21_TEST_NE[155],RN21_Map_NE[155]) ,MOV(RN21_TEST_NE[156],RN21_Map_NE[156]) ,MOV(RN21_TEST_NE[157],RN21_Map_NE[157]) ,MOV(RN21_TEST_NE[158],RN21_Map_NE[158]) ,MOV(RN21_TEST_NE[159],RN21_Map_NE[159]) ,MOV(RN21_TEST_NE[160],RN21_Map_NE[160]) ,MOV(RN21_TEST_NE[161],RN21_Map_NE[161]) ,MOV(RN21_TEST_NE[162],RN21_Map_NE[162]) ,MOV(RN21_TEST_NE[163],RN21_Map_NE[163]) ,MOV(RN21_TEST_NE[164],RN21_Map_NE[164]) ,MOV(RN21_TEST_NE[165],RN21_Map_NE[165]) ,MOV(RN21_TEST_NE[166],RN21_Map_NE[166]) ,MOV(RN21_TEST_NE[167],RN21_Map_NE[167]) ,MOV(RN21_TEST_NE[168],RN21_Map_NE[168]) ,MOV(RN21_TEST_NE[169],RN21_Map_NE[169]) ,MOV(RN21_TEST_NE[170],RN21_Map_NE[170]) ,MOV(RN21_TEST_NE[171],RN21_Map_NE[171]) ,MOV(RN21_TEST_NE[172],RN21_Map_NE[172]) ,MOV(RN21_TEST_NE[173],RN21_Map_NE[173]) ,MOV(RN21_TEST_NE[174],RN21_Map_NE[174]) ,MOV(RN21_TEST_NE[175],RN21_Map_NE[175]) ,MOV(RN21_TEST_NE[176],RN21_Map_NE[176]) ,MOV(RN21_TEST_NE[177],RN21_Map_NE[177]) ,MOV(RN21_TEST_NE[178],RN21_Map_NE[178]) ,MOV(RN21_TEST_NE[179],RN21_Map_NE[179]) ,MOV(RN21_TEST_NE[180],RN21_Map_NE[180]) ,MOV(RN21_TEST_NE[181],RN21_Map_NE[181]) ,MOV(RN21_TEST_NE[182],RN21_Map_NE[182]) ,MOV(RN21_TEST_NE[183],RN21_Map_NE[183]) ,MOV(RN21_TEST_NE[184],RN21_Map_NE[184]) ,MOV(RN21_TEST_NE[185],RN21_Map_NE[185]) ,MOV(RN21_TEST_NE[186],RN21_Map_NE[186]) ,MOV(RN21_TEST_NE[187],RN21_Map_NE[187]) ,MOV(RN21_TEST_NE[188],RN21_Map_NE[188]) ,MOV(RN21_TEST_NE[189],RN21_Map_NE[189]) ,MOV(RN21_TEST_NE[190],RN21_Map_NE[190]) ,MOV(RN21_TEST_NE[191],RN21_Map_NE[191]) ,MOV(RN21_TEST_NE[192],RN21_Map_NE[192]) ,MOV(RN21_TEST_NE[193],RN21_Map_NE[193]) ,MOV(RN21_TEST_NE[194],RN21_Map_NE[194]) ,MOV(RN21_TEST_NE[195],RN21_Map_NE[195]) ,MOV(RN21_TEST_NE[196],RN21_Map_NE[196]) ,MOV(RN21_TEST_NE[197],RN21_Map_NE[197]) ,MOV(RN21_TEST_NE[198],RN21_Map_NE[198]) ,MOV(RN21_TEST_NE[199],RN21_Map_NE[199]) ,MOV(RN21_TEST_NE[200],RN21_Map_NE[200]) ,MOV(RN21_TEST_NE[201],RN21_Map_NE[201]) ,MOV(RN21_TEST_NE[202],RN21_Map_NE[202]) ,MOV(RN21_TEST_NE[203],RN21_Map_NE[203]) ,MOV(RN21_TEST_NE[204],RN21_Map_NE[204]) ,MOV(RN21_TEST_NE[205],RN21_Map_NE[205]) ,MOV(RN21_TEST_NE[206],RN21_Map_NE[206]) ,MOV(RN21_TEST_NE[207],RN21_Map_NE[207]) ,MOV(RN21_TEST_NE[208],RN21_Map_NE[208]) ,MOV(RN21_TEST_NE[209],RN21_Map_NE[209]) ,MOV(RN21_TEST_NE[210],RN21_Map_NE[210]) ,MOV(RN21_TEST_NE[211],RN21_Map_NE[211]) ,MOV(RN21_TEST_NE[212],RN21_Map_NE[212]) ,MOV(RN21_TEST_NE[213],RN21_Map_NE[213]) ,MOV(RN21_TEST_NE[214],RN21_Map_NE[214]) ,MOV(RN21_TEST_NE[215],RN21_Map_NE[215]) ,MOV(RN21_TEST_NE[216],RN21_Map_NE[216]) ,MOV(RN21_TEST_NE[217],RN21_Map_NE[217]) ,MOV(RN21_TEST_NE[218],RN21_Map_NE[218]) ,MOV(RN21_TEST_NE[219],RN21_Map_NE[219]) ,MOV(RN21_TEST_NE[220],RN21_Map_NE[220]) ,MOV(RN21_TEST_NE[221],RN21_Map_NE[221]) ,MOV(RN21_TEST_NE[222],RN21_Map_NE[222]) ,MOV(RN21_TEST_NE[223],RN21_Map_NE[223]) ,MOV(RN21_TEST_NE[224],RN21_Map_NE[224]) ,MOV(RN21_TEST_NE[225],RN21_Map_NE[225]) ,MOV(RN21_TEST_NE[226],RN21_Map_NE[226]) ,MOV(RN21_TEST_NE[227],RN21_Map_NE[227]) ,MOV(RN21_TEST_NE[228],RN21_Map_NE[228]) ,MOV(RN21_TEST_NE[229],RN21_Map_NE[229]) ,MOV(RN21_TEST_NE[230],RN21_Map_NE[230]) ,MOV(RN21_TEST_NE[231],RN21_Map_NE[231]) ,MOV(RN21_TEST_NE[232],RN21_Map_NE[232]) ,MOV(RN21_TEST_NE[233],RN21_Map_NE[233]) ,MOV(RN21_TEST_NE[234],RN21_Map_NE[234]) ,MOV(RN21_TEST_NE[235],RN21_Map_NE[235]) ,MOV(RN21_TEST_NE[236],RN21_Map_NE[236]) ,MOV(RN21_TEST_NE[237],RN21_Map_NE[237]) ,MOV(RN21_TEST_NE[238],RN21_Map_NE[238]) ,MOV(RN21_TEST_NE[239],RN21_Map_NE[239]) ,MOV(RN21_TEST_NE[240],RN21_Map_NE[240]) ,MOV(RN21_TEST_NE[241],RN21_Map_NE[241]) ,MOV(RN21_TEST_NE[242],RN21_Map_NE[242]) ,MOV(RN21_TEST_NE[243],RN21_Map_NE[243]) ,MOV(RN21_TEST_NE[244],RN21_Map_NE[244]) ,MOV(RN21_TEST_NE[245],RN21_Map_NE[245]) ,MOV(RN21_TEST_NE[246],RN21_Map_NE[246]) ,MOV(RN21_TEST_NE[247],RN21_Map_NE[247]) ,MOV(RN21_TEST_NE[248],RN21_Map_NE[248]) ,MOV(RN21_TEST_NE[249],RN21_Map_NE[249]) ,MOV(RN21_TEST_NE[250],RN21_Map_NE[250]) ,MOV(RN21_TEST_NE[251],RN21_Map_NE[251]) ,MOV(RN21_TEST_NE[252],RN21_Map_NE[252]) ,MOV(RN21_TEST_NE[253],RN21_Map_NE[253]) ,MOV(RN21_TEST_NE[254],RN21_Map_NE[254]) ,MOV(RN21_TEST_NE[255],RN21_Map_NE[255]) ,MOV(RN21_TEST_NE[256],RN21_Map_NE[256]) ,MOV(RN21_TEST_NE[257],RN21_Map_NE[257]) ,MOV(RN21_TEST_NE[258],RN21_Map_NE[258]) ,MOV(RN21_TEST_NE[259],RN21_Map_NE[259]) ,MOV(RN21_TEST_NE[260],RN21_Map_NE[260]) ,MOV(RN21_TEST_NE[261],RN21_Map_NE[261]) ,MOV(RN21_TEST_NE[262],RN21_Map_NE[262]) ,MOV(RN21_TEST_NE[263],RN21_Map_NE[263]) ,MOV(RN21_TEST_NE[264],RN21_Map_NE[264]) ,MOV(RN21_TEST_NE[265],RN21_Map_NE[265]) ,MOV(RN21_TEST_NE[266],RN21_Map_NE[266]) ,MOV(RN21_TEST_NE[267],RN21_Map_NE[267]) ,MOV(RN21_TEST_NE[268],RN21_Map_NE[268]) ,MOV(RN21_TEST_NE[269],RN21_Map_NE[269]) ,MOV(RN21_TEST_NE[270],RN21_Map_NE[270]) ,MOV(RN21_TEST_NE[271],RN21_Map_NE[271]) ,MOV(RN21_TEST_NE[272],RN21_Map_NE[272]) ,MOV(RN21_TEST_NE[273],RN21_Map_NE[273]) ,MOV(RN21_TEST_NE[274],RN21_Map_NE[274]) ,MOV(RN21_TEST_NE[275],RN21_Map_NE[275]) ,MOV(RN21_TEST_NE[276],RN21_Map_NE[276]) ,MOV(RN21_TEST_NE[277],RN21_Map_NE[277]) ,MOV(RN21_TEST_NE[278],RN21_Map_NE[278]) ,MOV(RN21_TEST_NE[279],RN21_Map_NE[279]) ,MOV(RN21_TEST_NE[280],RN21_Map_NE[280]) ,MOV(RN21_TEST_NE[281],RN21_Map_NE[281]) ,MOV(RN21_TEST_NE[282],RN21_Map_NE[282]) ,MOV(RN21_TEST_NE[283],RN21_Map_NE[283]) ,MOV(RN21_TEST_NE[284],RN21_Map_NE[284]) ,MOV(RN21_TEST_NE[285],RN21_Map_NE[285]) ,MOV(RN21_TEST_NE[286],RN21_Map_NE[286]) ,MOV(RN21_TEST_NE[287],RN21_Map_NE[287]) ,MOV(RN21_TEST_NE[288],RN21_Map_NE[288]) ,MOV(RN21_TEST_NE[289],RN21_Map_NE[289]) ,MOV(RN21_TEST_NE[290],RN21_Map_NE[290]) ,MOV(RN21_TEST_NE[291],RN21_Map_NE[291]) ,MOV(RN21_TEST_NE[292],RN21_Map_NE[292]) ,MOV(RN21_TEST_NE[293],RN21_Map_NE[293]) ,MOV(RN21_TEST_NE[294],RN21_Map_NE[294]) ,MOV(RN21_TEST_NE[295],RN21_Map_NE[295]) ,MOV(RN21_TEST_NE[296],RN21_Map_NE[296]) ,MOV(RN21_TEST_NE[297],RN21_Map_NE[297]) ,MOV(RN21_TEST_NE[298],RN21_Map_NE[298]) ,MOV(RN21_TEST_NE[299],RN21_Map_NE[299]) ,MOV(RN21_TEST_NE[300],RN21_Map_NE[300]) ];
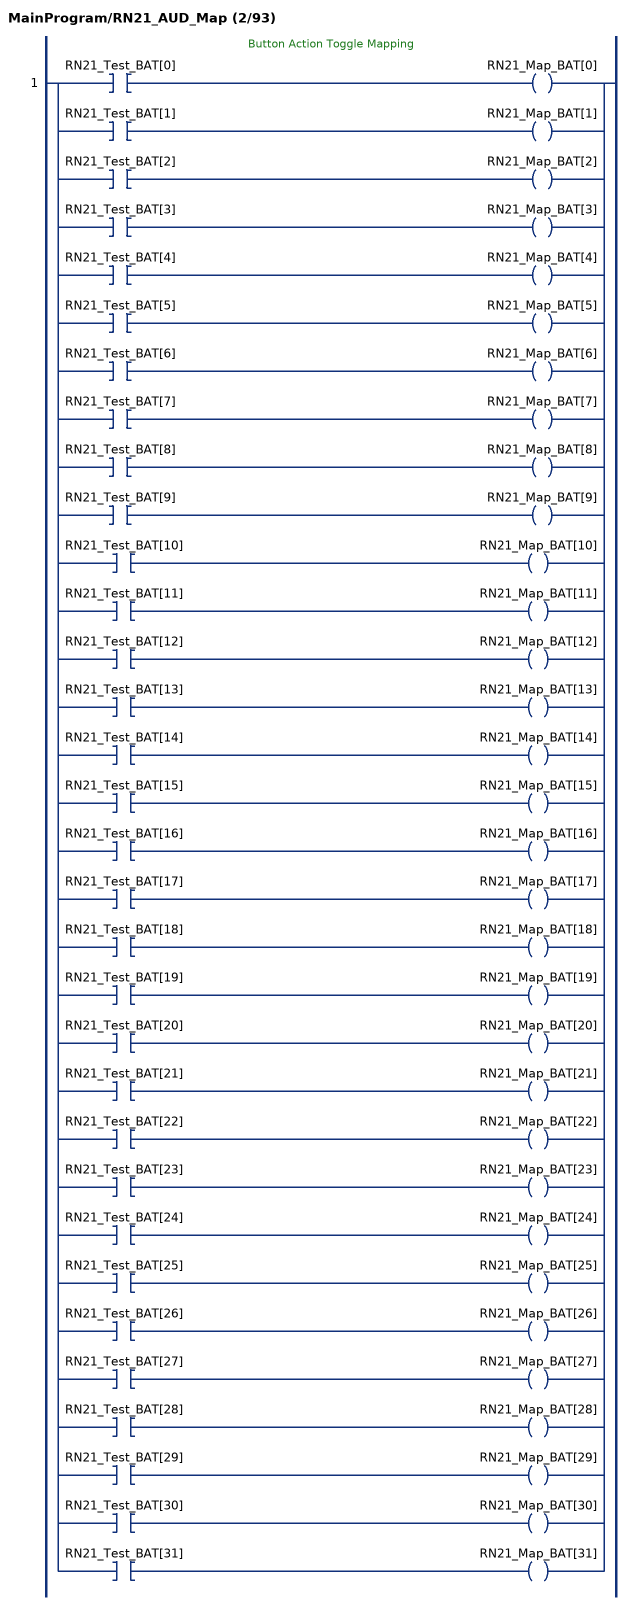
   // Button Action Toggle Mapping
   1: [XIC(RN21_Test_BAT[0]) OTE(RN21_Map_BAT[0]) ,XIC(RN21_Test_BAT[1]) OTE(RN21_Map_BAT[1]) ,XIC(RN21_Test_BAT[2]) OTE(RN21_Map_BAT[2]) ,XIC(RN21_Test_BAT[3]) OTE(RN21_Map_BAT[3]) ,XIC(RN21_Test_BAT[4]) OTE(RN21_Map_BAT[4]) ,XIC(RN21_Test_BAT[5]) OTE(RN21_Map_BAT[5]) ,XIC(RN21_Test_BAT[6]) OTE(RN21_Map_BAT[6]) ,XIC(RN21_Test_BAT[7]) OTE(RN21_Map_BAT[7]) ,XIC(RN21_Test_BAT[8]) OTE(RN21_Map_BAT[8]) ,XIC(RN21_Test_BAT[9]) OTE(RN21_Map_BAT[9]) ,XIC(RN21_Test_BAT[10]) OTE(RN21_Map_BAT[10]) ,XIC(RN21_Test_BAT[11]) OTE(RN21_Map_BAT[11]) ,XIC(RN21_Test_BAT[12]) OTE(RN21_Map_BAT[12]) ,XIC(RN21_Test_BAT[13]) OTE(RN21_Map_BAT[13]) ,XIC(RN21_Test_BAT[14]) OTE(RN21_Map_BAT[14]) ,XIC(RN21_Test_BAT[15]) OTE(RN21_Map_BAT[15]) ,XIC(RN21_Test_BAT[16]) OTE(RN21_Map_BAT[16]) ,XIC(RN21_Test_BAT[17]) OTE(RN21_Map_BAT[17]) ,XIC(RN21_Test_BAT[18]) OTE(RN21_Map_BAT[18]) ,XIC(RN21_Test_BAT[19]) OTE(RN21_Map_BAT[19]) ,XIC(RN21_Test_BAT[20]) OTE(RN21_Map_BAT[20]) ,XIC(RN21_Test_BAT[21]) OTE(RN21_Map_BAT[21]) ,XIC(RN21_Test_BAT[22]) OTE(RN21_Map_BAT[22]) ,XIC(RN21_Test_BAT[23]) OTE(RN21_Map_BAT[23]) ,XIC(RN21_Test_BAT[24]) OTE(RN21_Map_BAT[24]) ,XIC(RN21_Test_BAT[25]) OTE(RN21_Map_BAT[25]) ,XIC(RN21_Test_BAT[26]) OTE(RN21_Map_BAT[26]) ,XIC(RN21_Test_BAT[27]) OTE(RN21_Map_BAT[27]) ,XIC(RN21_Test_BAT[28]) OTE(RN21_Map_BAT[28]) ,XIC(RN21_Test_BAT[29]) OTE(RN21_Map_BAT[29]) ,XIC(RN21_Test_BAT[30]) OTE(RN21_Map_BAT[30]) ,XIC(RN21_Test_BAT[31]) OTE(RN21_Map_BAT[31]) ];
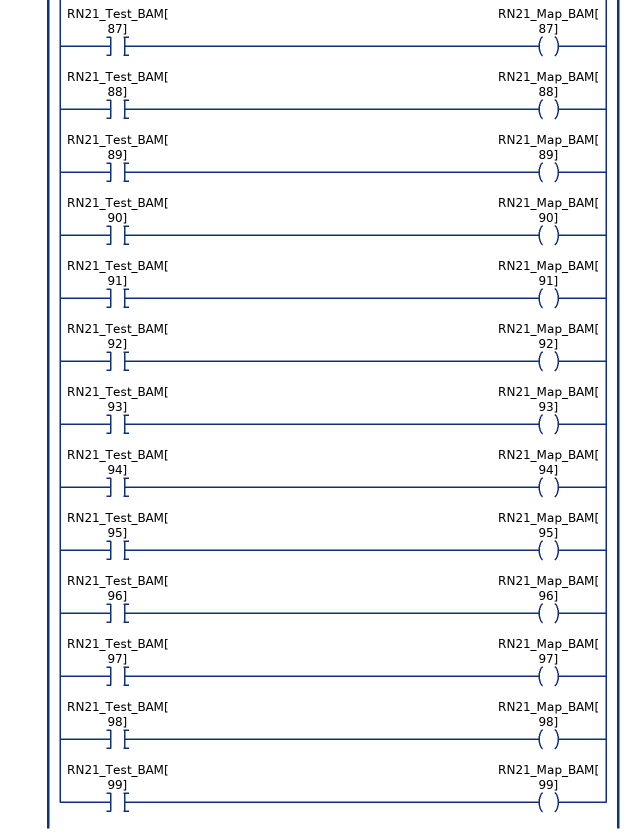
   // Button Action Momentary Mapping
   2: [XIC(RN21_Test_BAM[0]) OTE(RN21_Map_BAM[0]) ,XIC(RN21_Test_BAM[1]) OTE(RN21_Map_BAM[1]) ,XIC(RN21_Test_BAM[2]) OTE(RN21_Map_BAM[2]) ,XIC(RN21_Test_BAM[3]) OTE(RN21_Map_BAM[3]) ,XIC(RN21_Test_BAM[4]) OTE(RN21_Map_BAM[4]) ,XIC(RN21_Test_BAM[5]) OTE(RN21_Map_BAM[5]) ,XIC(RN21_Test_BAM[6]) OTE(RN21_Map_BAM[6]) ,XIC(RN21_Test_BAM[7]) OTE(RN21_Map_BAM[7]) ,XIC(RN21_Test_BAM[8]) OTE(RN21_Map_BAM[8]) ,XIC(RN21_Test_BAM[9]) OTE(RN21_Map_BAM[9]) ,XIC(RN21_Test_BAM[10]) OTE(RN21_Map_BAM[10]) ,XIC(RN21_Test_BAM[11]) OTE(RN21_Map_BAM[11]) ,XIC(RN21_Test_BAM[12]) OTE(RN21_Map_BAM[12]) ,XIC(RN21_Test_BAM[13]) OTE(RN21_Map_BAM[13]) ,XIC(RN21_Test_BAM[14]) OTE(RN21_Map_BAM[14]) ,XIC(RN21_Test_BAM[15]) OTE(RN21_Map_BAM[15]) ,XIC(RN21_Test_BAM[16]) OTE(RN21_Map_BAM[16]) ,XIC(RN21_Test_BAM[17]) OTE(RN21_Map_BAM[17]) ,XIC(RN21_Test_BAM[18]) OTE(RN21_Map_BAM[18]) ,XIC(RN21_Test_BAM[19]) OTE(RN21_Map_BAM[19]) ,XIC(RN21_Test_BAM[20]) OTE(RN21_Map_BAM[20]) ,XIC(RN21_Test_BAM[21]) OTE(RN21_Map_BAM[21]) ,XIC(RN21_Test_BAM[22]) OTE(RN21_Map_BAM[22]) ,XIC(RN21_Test_BAM[23]) OTE(RN21_Map_BAM[23]) ,XIC(RN21_Test_BAM[24]) OTE(RN21_Map_BAM[24]) ,XIC(RN21_Test_BAM[25]) OTE(RN21_Map_BAM[25]) ,XIC(RN21_Test_BAM[26]) OTE(RN21_Map_BAM[26]) ,XIC(RN21_Test_BAM[27]) OTE(RN21_Map_BAM[27]) ,XIC(RN21_Test_BAM[28]) OTE(RN21_Map_BAM[28]) ,XIC(RN21_Test_BAM[29]) OTE(RN21_Map_BAM[29]) ,XIC(RN21_Test_BAM[30]) OTE(RN21_Map_BAM[30]) ,XIC(RN21_Test_BAM[31]) OTE(RN21_Map_BAM[31]) ,XIC(RN21_Test_BAM[32]) OTE(RN21_Map_BAM[32]) ,XIC(RN21_Test_BAM[33]) OTE(RN21_Map_BAM[33]) ,XIC(RN21_Test_BAM[34]) OTE(RN21_Map_BAM[34]) ,XIC(RN21_Test_BAM[35]) OTE(RN21_Map_BAM[35]) ,XIC(RN21_Test_BAM[36]) OTE(RN21_Map_BAM[36]) ,XIC(RN21_Test_BAM[37]) OTE(RN21_Map_BAM[37]) ,XIC(RN21_Test_BAM[38]) OTE(RN21_Map_BAM[38]) ,XIC(RN21_Test_BAM[39]) OTE(RN21_Map_BAM[39]) ,XIC(RN21_Test_BAM[40]) OTE(RN21_Map_BAM[40]) ,XIC(RN21_Test_BAM[41]) OTE(RN21_Map_BAM[41]) ,XIC(RN21_Test_BAM[42]) OTE(RN21_Map_BAM[42]) ,XIC(RN21_Test_BAM[43]) OTE(RN21_Map_BAM[43]) ,XIC(RN21_Test_BAM[44]) OTE(RN21_Map_BAM[44]) ,XIC(RN21_Test_BAM[45]) OTE(RN21_Map_BAM[45]) ,XIC(RN21_Test_BAM[46]) OTE(RN21_Map_BAM[46]) ,XIC(RN21_Test_BAM[47]) OTE(RN21_Map_BAM[47]) ,XIC(RN21_Test_BAM[48]) OTE(RN21_Map_BAM[48]) ,XIC(RN21_Test_BAM[49]) OTE(RN21_Map_BAM[49]) ,XIC(RN21_Test_BAM[50]) OTE(RN21_Map_BAM[50]) ,XIC(RN21_Test_BAM[51]) OTE(RN21_Map_BAM[51]) ,XIC(RN21_Test_BAM[52]) OTE(RN21_Map_BAM[52]) ,XIC(RN21_Test_BAM[53]) OTE(RN21_Map_BAM[53]) ,XIC(RN21_Test_BAM[54]) OTE(RN21_Map_BAM[54]) ,XIC(RN21_Test_BAM[55]) OTE(RN21_Map_BAM[55]) ,XIC(RN21_Test_BAM[56]) OTE(RN21_Map_BAM[56]) ,XIC(RN21_Test_BAM[57]) OTE(RN21_Map_BAM[57]) ,XIC(RN21_Test_BAM[58]) OTE(RN21_Map_BAM[58]) ,XIC(RN21_Test_BAM[59]) OTE(RN21_Map_BAM[59]) ,XIC(RN21_Test_BAM[60]) OTE(RN21_Map_BAM[60]) ,XIC(RN21_Test_BAM[61]) OTE(RN21_Map_BAM[61]) ,XIC(RN21_Test_BAM[62]) OTE(RN21_Map_BAM[62]) ,XIC(RN21_Test_BAM[63]) OTE(RN21_Map_BAM[63]) ,XIC(RN21_Test_BAM[64]) OTE(RN21_Map_BAM[64]) ,XIC(RN21_Test_BAM[65]) OTE(RN21_Map_BAM[65]) ,XIC(RN21_Test_BAM[66]) OTE(RN21_Map_BAM[66]) ,XIC(RN21_Test_BAM[67]) OTE(RN21_Map_BAM[67]) ,XIC(RN21_Test_BAM[68]) OTE(RN21_Map_BAM[68]) ,XIC(RN21_Test_BAM[69]) OTE(RN21_Map_BAM[69]) ,XIC(RN21_Test_BAM[70]) OTE(RN21_Map_BAM[70]) ,XIC(RN21_Test_BAM[71]) OTE(RN21_Map_BAM[71]) ,XIC(RN21_Test_BAM[72]) OTE(RN21_Map_BAM[72]) ,XIC(RN21_Test_BAM[73]) OTE(RN21_Map_BAM[73]) ,XIC(RN21_Test_BAM[74]) OTE(RN21_Map_BAM[74]) ,XIC(RN21_Test_BAM[75]) OTE(RN21_Map_BAM[75]) ,XIC(RN21_Test_BAM[76]) OTE(RN21_Map_BAM[76]) ,XIC(RN21_Test_BAM[77]) OTE(RN21_Map_BAM[77]) ,XIC(RN21_Test_BAM[78]) OTE(RN21_Map_BAM[78]) ,XIC(RN21_Test_BAM[79]) OTE(RN21_Map_BAM[79]) ,XIC(RN21_Test_BAM[80]) OTE(RN21_Map_BAM[80]) ,XIC(RN21_Test_BAM[81]) OTE(RN21_Map_BAM[81]) ,XIC(RN21_Test_BAM[82]) OTE(RN21_Map_BAM[82]) ,XIC(RN21_Test_BAM[83]) OTE(RN21_Map_BAM[83]) ,XIC(RN21_Test_BAM[84]) OTE(RN21_Map_BAM[84]) ,XIC(RN21_Test_BAM[85]) OTE(RN21_Map_BAM[85]) ,XIC(RN21_Test_BAM[86]) OTE(RN21_Map_BAM[86]) ,XIC(RN21_Test_BAM[87]) OTE(RN21_Map_BAM[87]) ,XIC(RN21_Test_BAM[88]) OTE(RN21_Map_BAM[88]) ,XIC(RN21_Test_BAM[89]) OTE(RN21_Map_BAM[89]) ,XIC(RN21_Test_BAM[90]) OTE(RN21_Map_BAM[90]) ,XIC(RN21_Test_BAM[91]) OTE(RN21_Map_BAM[91]) ,XIC(RN21_Test_BAM[92]) OTE(RN21_Map_BAM[92]) ,XIC(RN21_Test_BAM[93]) OTE(RN21_Map_BAM[93]) ,XIC(RN21_Test_BAM[94]) OTE(RN21_Map_BAM[94]) ,XIC(RN21_Test_BAM[95]) OTE(RN21_Map_BAM[95]) ,XIC(RN21_Test_BAM[96]) OTE(RN21_Map_BAM[96]) ,XIC(RN21_Test_BAM[97]) OTE(RN21_Map_BAM[97]) ,XIC(RN21_Test_BAM[98]) OTE(RN21_Map_BAM[98]) ,XIC(RN21_Test_BAM[99]) OTE(RN21_Map_BAM[99]) ];
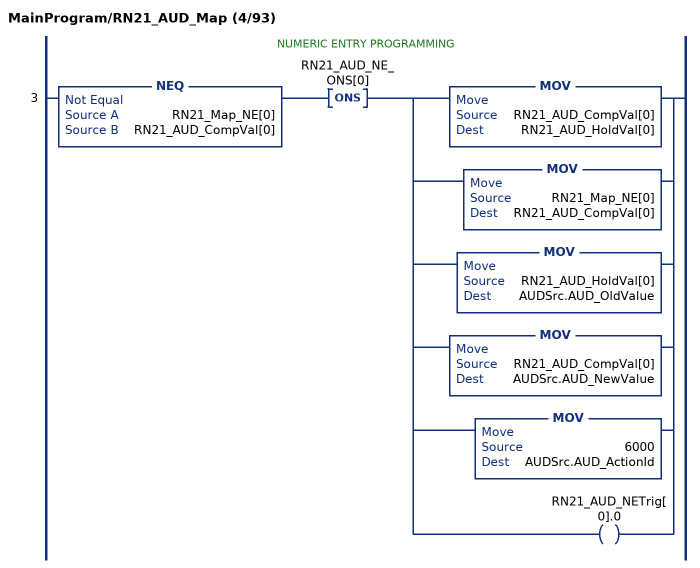
   // NUMERIC ENTRY PROGRAMMING
   3: NEQ(RN21_Map_NE[0],RN21_AUD_CompVal[0])ONS(RN21_AUD_NE_ONS[0])[MOV(RN21_AUD_CompVal[0],RN21_AUD_HoldVal[0]) ,MOV(RN21_Map_NE[0],RN21_AUD_CompVal[0]) ,MOV(RN21_AUD_HoldVal[0],AUDSrc.AUD_OldValue) ,MOV(RN21_AUD_CompVal[0],AUDSrc.AUD_NewValue) ,MOV(6000,AUDSrc.AUD_ActionId) ,OTE(RN21_AUD_NETrig[0].0) ];
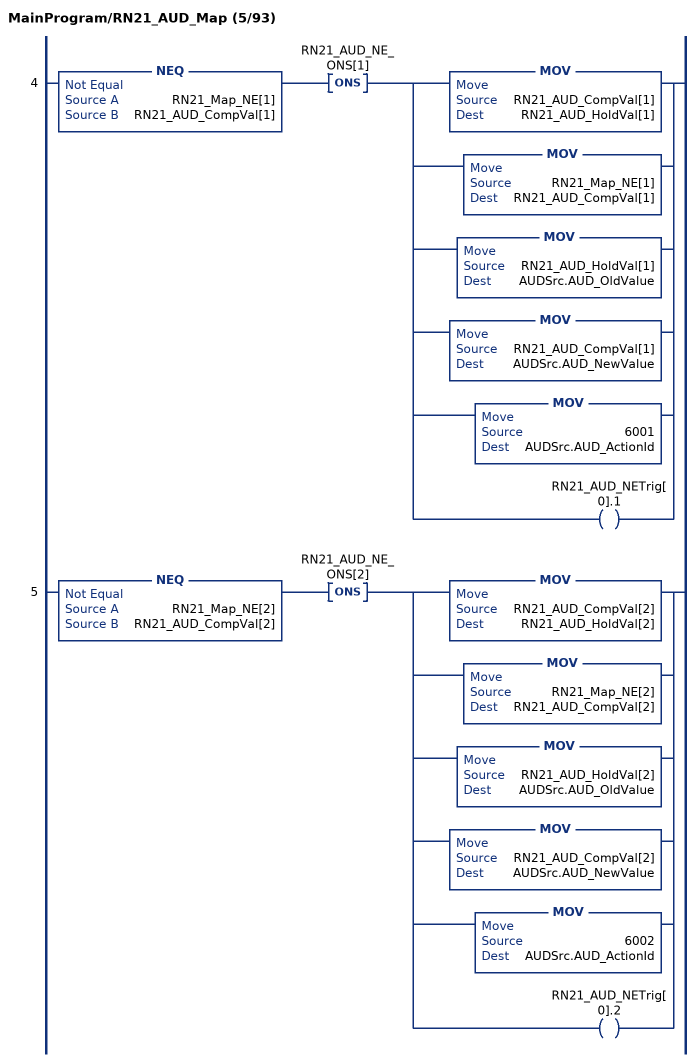
   4: NEQ(RN21_Map_NE[1],RN21_AUD_CompVal[1])ONS(RN21_AUD_NE_ONS[1])[MOV(RN21_AUD_CompVal[1],RN21_AUD_HoldVal[1]) ,MOV(RN21_Map_NE[1],RN21_AUD_CompVal[1]) ,MOV(RN21_AUD_HoldVal[1],AUDSrc.AUD_OldValue) ,MOV(RN21_AUD_CompVal[1],AUDSrc.AUD_NewValue) ,MOV(6001,AUDSrc.AUD_ActionId) ,OTE(RN21_AUD_NETrig[0].1) ];
   5: NEQ(RN21_Map_NE[2],RN21_AUD_CompVal[2])ONS(RN21_AUD_NE_ONS[2])[MOV(RN21_AUD_CompVal[2],RN21_AUD_HoldVal[2]) ,MOV(RN21_Map_NE[2],RN21_AUD_CompVal[2]) ,MOV(RN21_AUD_HoldVal[2],AUDSrc.AUD_OldValue) ,MOV(RN21_AUD_CompVal[2],AUDSrc.AUD_NewValue) ,MOV(6002,AUDSrc.AUD_ActionId) ,OTE(RN21_AUD_NETrig[0].2) ];
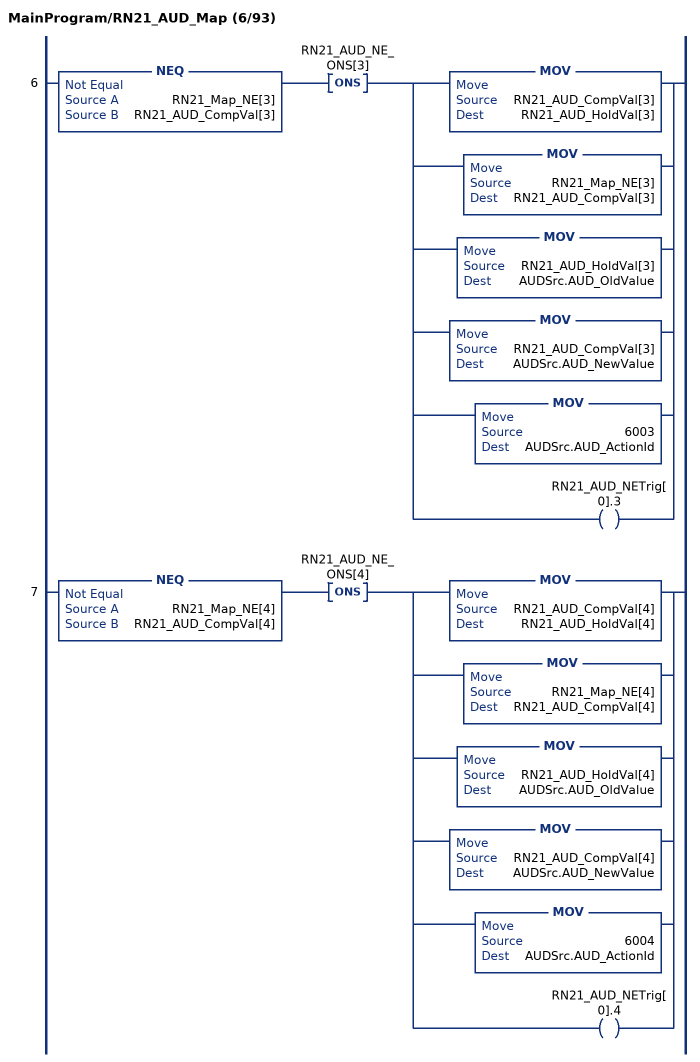
   6: NEQ(RN21_Map_NE[3],RN21_AUD_CompVal[3])ONS(RN21_AUD_NE_ONS[3])[MOV(RN21_AUD_CompVal[3],RN21_AUD_HoldVal[3]) ,MOV(RN21_Map_NE[3],RN21_AUD_CompVal[3]) ,MOV(RN21_AUD_HoldVal[3],AUDSrc.AUD_OldValue) ,MOV(RN21_AUD_CompVal[3],AUDSrc.AUD_NewValue) ,MOV(6003,AUDSrc.AUD_ActionId) ,OTE(RN21_AUD_NETrig[0].3) ];
   7: NEQ(RN21_Map_NE[4],RN21_AUD_CompVal[4])ONS(RN21_AUD_NE_ONS[4])[MOV(RN21_AUD_CompVal[4],RN21_AUD_HoldVal[4]) ,MOV(RN21_Map_NE[4],RN21_AUD_CompVal[4]) ,MOV(RN21_AUD_HoldVal[4],AUDSrc.AUD_OldValue) ,MOV(RN21_AUD_CompVal[4],AUDSrc.AUD_NewValue) ,MOV(6004,AUDSrc.AUD_ActionId) ,OTE(RN21_AUD_NETrig[0].4) ];
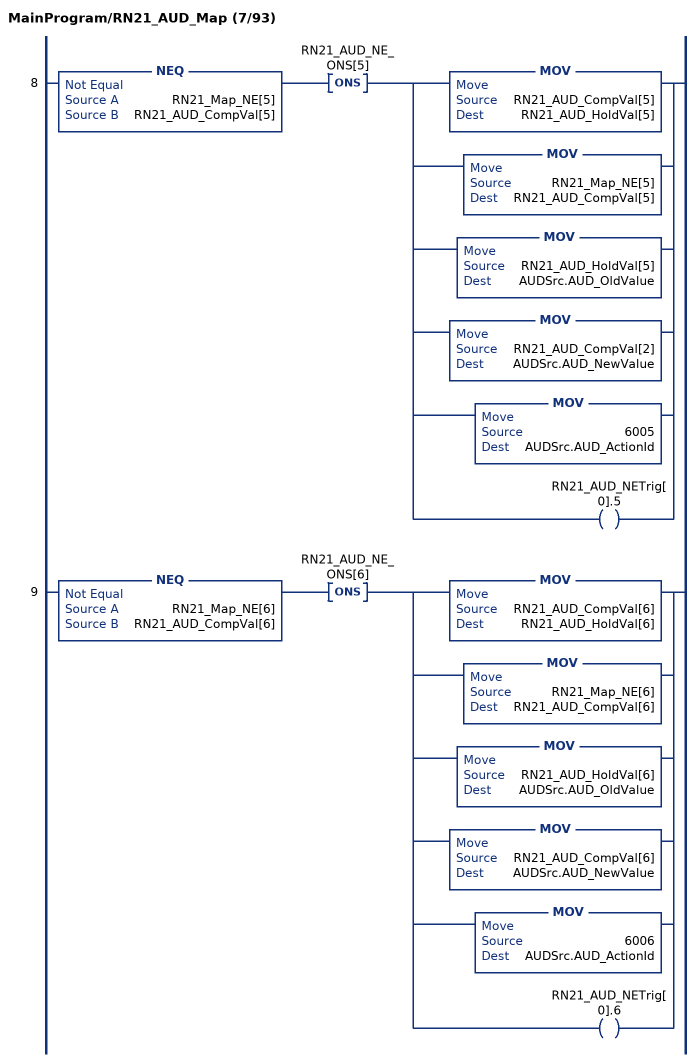
   8: NEQ(RN21_Map_NE[5],RN21_AUD_CompVal[5])ONS(RN21_AUD_NE_ONS[5])[MOV(RN21_AUD_CompVal[5],RN21_AUD_HoldVal[5]) ,MOV(RN21_Map_NE[5],RN21_AUD_CompVal[5]) ,MOV(RN21_AUD_HoldVal[5],AUDSrc.AUD_OldValue) ,MOV(RN21_AUD_CompVal[2],AUDSrc.AUD_NewValue) ,MOV(6005,AUDSrc.AUD_ActionId) ,OTE(RN21_AUD_NETrig[0].5) ];
   9: NEQ(RN21_Map_NE[6],RN21_AUD_CompVal[6])ONS(RN21_AUD_NE_ONS[6])[MOV(RN21_AUD_CompVal[6],RN21_AUD_HoldVal[6]) ,MOV(RN21_Map_NE[6],RN21_AUD_CompVal[6]) ,MOV(RN21_AUD_HoldVal[6],AUDSrc.AUD_OldValue) ,MOV(RN21_AUD_CompVal[6],AUDSrc.AUD_NewValue) ,MOV(6006,AUDSrc.AUD_ActionId) ,OTE(RN21_AUD_NETrig[0].6) ];
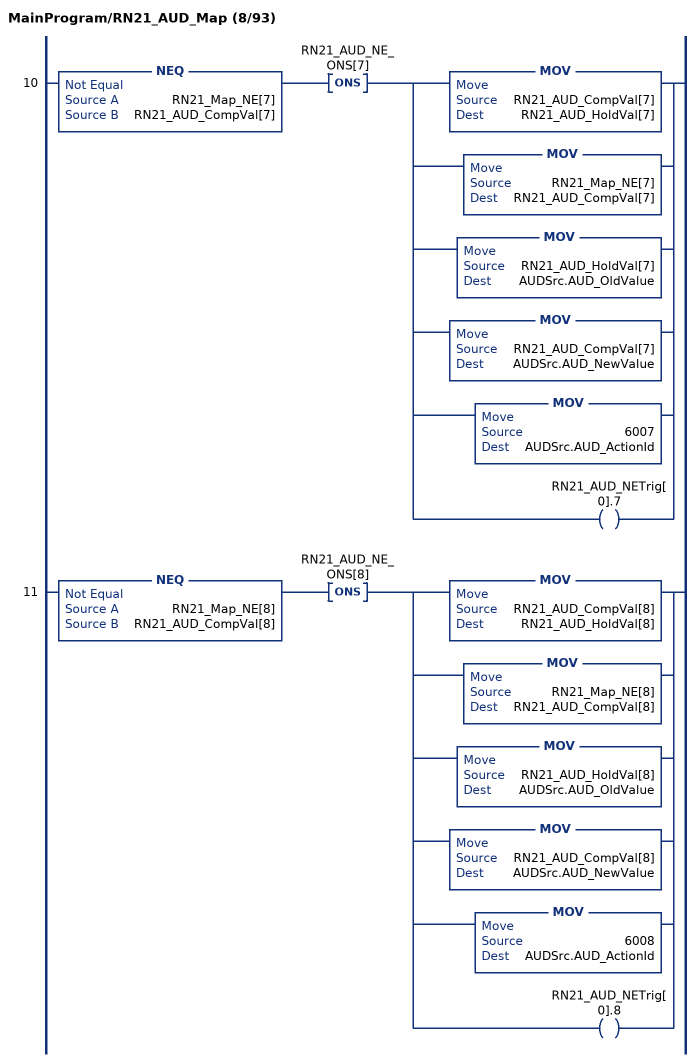
   10: NEQ(RN21_Map_NE[7],RN21_AUD_CompVal[7])ONS(RN21_AUD_NE_ONS[7])[MOV(RN21_AUD_CompVal[7],RN21_AUD_HoldVal[7]) ,MOV(RN21_Map_NE[7],RN21_AUD_CompVal[7]) ,MOV(RN21_AUD_HoldVal[7],AUDSrc.AUD_OldValue) ,MOV(RN21_AUD_CompVal[7],AUDSrc.AUD_NewValue) ,MOV(6007,AUDSrc.AUD_ActionId) ,OTE(RN21_AUD_NETrig[0].7) ];
   11: NEQ(RN21_Map_NE[8],RN21_AUD_CompVal[8])ONS(RN21_AUD_NE_ONS[8])[MOV(RN21_AUD_CompVal[8],RN21_AUD_HoldVal[8]) ,MOV(RN21_Map_NE[8],RN21_AUD_CompVal[8]) ,MOV(RN21_AUD_HoldVal[8],AUDSrc.AUD_OldValue) ,MOV(RN21_AUD_CompVal[8],AUDSrc.AUD_NewValue) ,MOV(6008,AUDSrc.AUD_ActionId) ,OTE(RN21_AUD_NETrig[0].8) ];
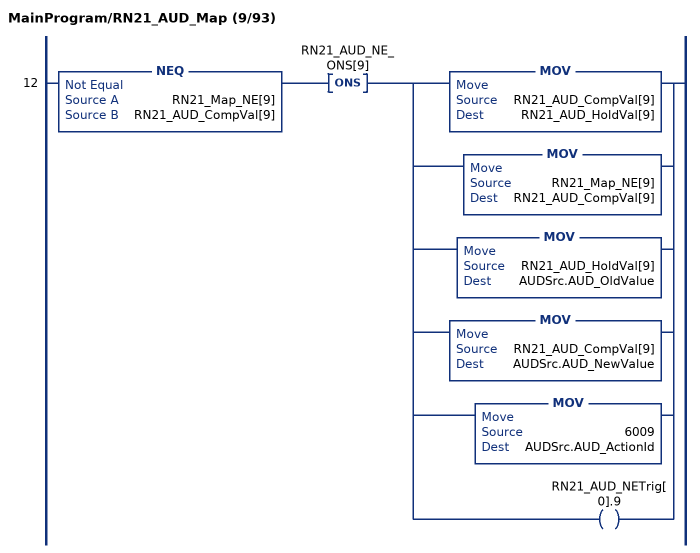
   12: NEQ(RN21_Map_NE[9],RN21_AUD_CompVal[9])ONS(RN21_AUD_NE_ONS[9])[MOV(RN21_AUD_CompVal[9],RN21_AUD_HoldVal[9]) ,MOV(RN21_Map_NE[9],RN21_AUD_CompVal[9]) ,MOV(RN21_AUD_HoldVal[9],AUDSrc.AUD_OldValue) ,MOV(RN21_AUD_CompVal[9],AUDSrc.AUD_NewValue) ,MOV(6009,AUDSrc.AUD_ActionId) ,OTE(RN21_AUD_NETrig[0].9) ];
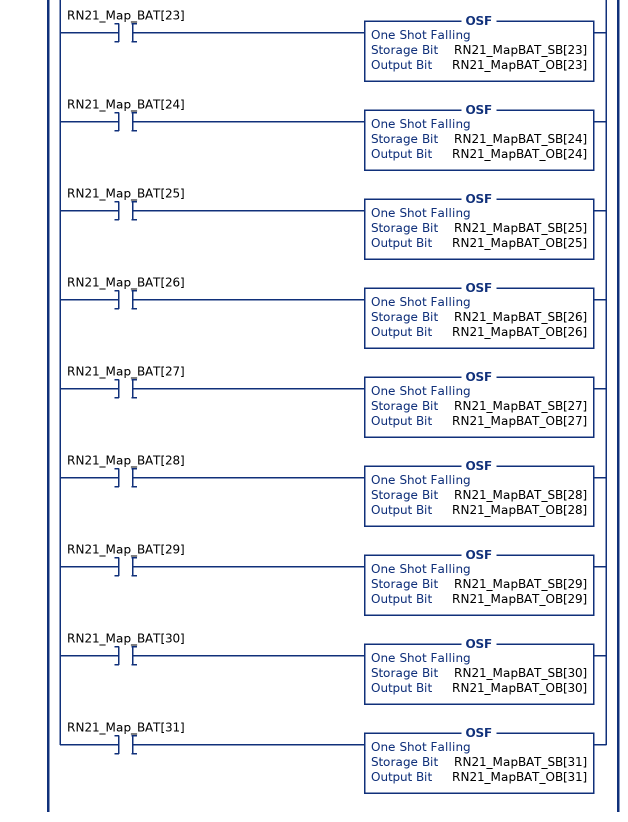
   13: [XIC(RN21_Map_BAT[0]) OSF(RN21_MapBAT_SB[0],RN21_MapBAT_OB[0]) ,XIC(RN21_Map_BAT[1]) OSF(RN21_MapBAT_SB[1],RN21_MapBAT_OB[1]) ,XIC(RN21_Map_BAT[2]) OSF(RN21_MapBAT_SB[2],RN21_MapBAT_OB[2]) ,XIC(RN21_Map_BAT[3]) OSF(RN21_MapBAT_SB[3],RN21_MapBAT_OB[3]) ,XIC(RN21_Map_BAT[4]) OSF(RN21_MapBAT_SB[4],RN21_MapBAT_OB[4]) ,XIC(RN21_Map_BAT[5]) OSF(RN21_MapBAT_SB[5],RN21_MapBAT_OB[5]) ,XIC(RN21_Map_BAT[6]) OSF(RN21_MapBAT_SB[6],RN21_MapBAT_OB[6]) ,XIC(RN21_Map_BAT[7]) OSF(RN21_MapBAT_SB[7],RN21_MapBAT_OB[7]) ,XIC(RN21_Map_BAT[8]) OSF(RN21_MapBAT_SB[8],RN21_MapBAT_OB[8]) ,XIC(RN21_Map_BAT[9]) OSF(RN21_MapBAT_SB[9],RN21_MapBAT_OB[9]) ,XIC(RN21_Map_BAT[10]) OSF(RN21_MapBAT_SB[10],RN21_MapBAT_OB[10]) ,XIC(RN21_Map_BAT[11]) OSF(RN21_MapBAT_SB[11],RN21_MapBAT_OB[11]) ,XIC(RN21_Map_BAT[12]) OSF(RN21_MapBAT_SB[12],RN21_MapBAT_OB[12]) ,XIC(RN21_Map_BAT[13]) OSF(RN21_MapBAT_SB[13],RN21_MapBAT_OB[13]) ,XIC(RN21_Map_BAT[14]) OSF(RN21_MapBAT_SB[14],RN21_MapBAT_OB[14]) ,XIC(RN21_Map_BAT[15]) OSF(RN21_MapBAT_SB[15],RN21_MapBAT_OB[15]) ,XIC(RN21_Map_BAT[16]) OSF(RN21_MapBAT_SB[16],RN21_MapBAT_OB[16]) ,XIC(RN21_Map_BAT[17]) OSF(RN21_MapBAT_SB[17],RN21_MapBAT_OB[17]) ,XIC(RN21_Map_BAT[18]) OSF(RN21_MapBAT_SB[18],RN21_MapBAT_OB[18]) ,XIC(RN21_Map_BAT[19]) OSF(RN21_MapBAT_SB[19],RN21_MapBAT_OB[19]) ,XIC(RN21_Map_BAT[20]) OSF(RN21_MapBAT_SB[20],RN21_MapBAT_OB[20]) ,XIC(RN21_Map_BAT[21]) OSF(RN21_MapBAT_SB[21],RN21_MapBAT_OB[21]) ,XIC(RN21_Map_BAT[22]) OSF(RN21_MapBAT_SB[22],RN21_MapBAT_OB[22]) ,XIC(RN21_Map_BAT[23]) OSF(RN21_MapBAT_SB[23],RN21_MapBAT_OB[23]) ,XIC(RN21_Map_BAT[24]) OSF(RN21_MapBAT_SB[24],RN21_MapBAT_OB[24]) ,XIC(RN21_Map_BAT[25]) OSF(RN21_MapBAT_SB[25],RN21_MapBAT_OB[25]) ,XIC(RN21_Map_BAT[26]) OSF(RN21_MapBAT_SB[26],RN21_MapBAT_OB[26]) ,XIC(RN21_Map_BAT[27]) OSF(RN21_MapBAT_SB[27],RN21_MapBAT_OB[27]) ,XIC(RN21_Map_BAT[28]) OSF(RN21_MapBAT_SB[28],RN21_MapBAT_OB[28]) ,XIC(RN21_Map_BAT[29]) OSF(RN21_MapBAT_SB[29],RN21_MapBAT_OB[29]) ,XIC(RN21_Map_BAT[30]) OSF(RN21_MapBAT_SB[30],RN21_MapBAT_OB[30]) ,XIC(RN21_Map_BAT[31]) OSF(RN21_MapBAT_SB[31],RN21_MapBAT_OB[31]) ];
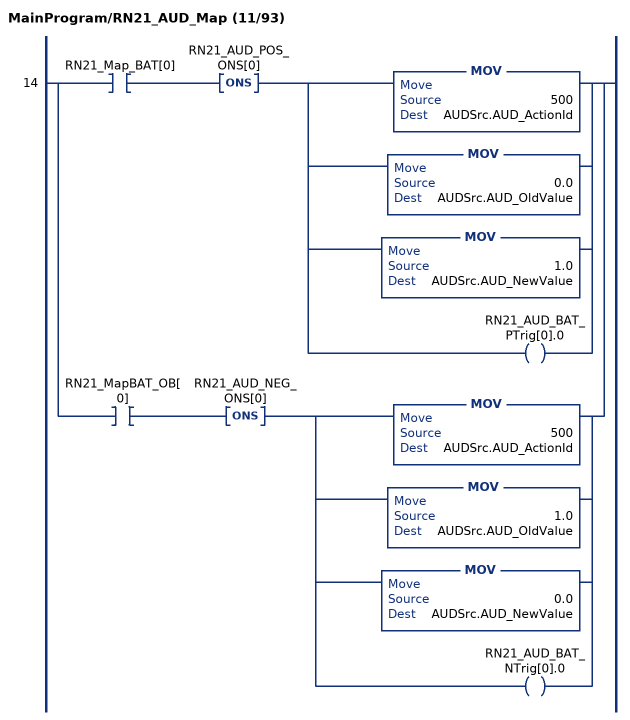
   14: [XIC(RN21_Map_BAT[0]) ONS(RN21_AUD_POS_ONS[0]) [MOV(500,AUDSrc.AUD_ActionId) ,MOV(0.0,AUDSrc.AUD_OldValue) ,MOV(1.0,AUDSrc.AUD_NewValue) ,OTE(RN21_AUD_BAT_PTrig[0].0) ] ,XIC(RN21_MapBAT_OB[0]) ONS(RN21_AUD_NEG_ONS[0]) [MOV(500,AUDSrc.AUD_ActionId) ,MOV(1.0,AUDSrc.AUD_OldValue) ,MOV(0.0,AUDSrc.AUD_NewValue) ,OTE(RN21_AUD_BAT_NTrig[0].0) ] ];
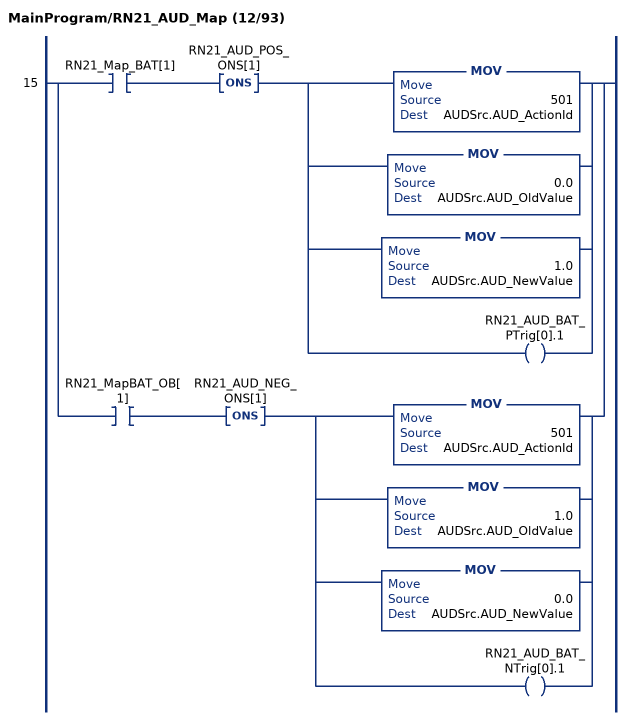
   15: [XIC(RN21_Map_BAT[1]) ONS(RN21_AUD_POS_ONS[1]) [MOV(501,AUDSrc.AUD_ActionId) ,MOV(0.0,AUDSrc.AUD_OldValue) ,MOV(1.0,AUDSrc.AUD_NewValue) ,OTE(RN21_AUD_BAT_PTrig[0].1) ] ,XIC(RN21_MapBAT_OB[1]) ONS(RN21_AUD_NEG_ONS[1]) [MOV(501,AUDSrc.AUD_ActionId) ,MOV(1.0,AUDSrc.AUD_OldValue) ,MOV(0.0,AUDSrc.AUD_NewValue) ,OTE(RN21_AUD_BAT_NTrig[0].1) ] ];
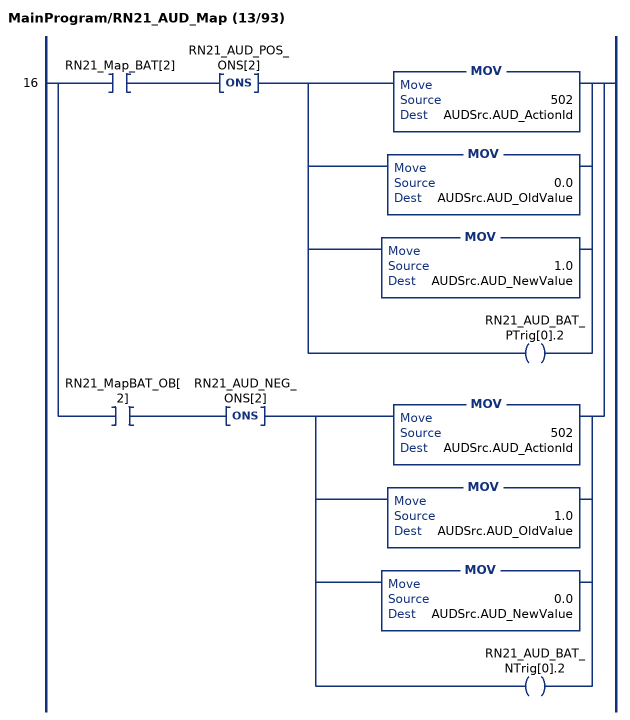
   16: [XIC(RN21_Map_BAT[2]) ONS(RN21_AUD_POS_ONS[2]) [MOV(502,AUDSrc.AUD_ActionId) ,MOV(0.0,AUDSrc.AUD_OldValue) ,MOV(1.0,AUDSrc.AUD_NewValue) ,OTE(RN21_AUD_BAT_PTrig[0].2) ] ,XIC(RN21_MapBAT_OB[2]) ONS(RN21_AUD_NEG_ONS[2]) [MOV(502,AUDSrc.AUD_ActionId) ,MOV(1.0,AUDSrc.AUD_OldValue) ,MOV(0.0,AUDSrc.AUD_NewValue) ,OTE(RN21_AUD_BAT_NTrig[0].2) ] ];
